LIN {X 0,Y 439.168,Z 450.878,A -85,B 0,C 180,E1 8974.952,E2 8974.952} C_VEL
LIN {X 0,Y 436.814,Z 482.203,A -85,B 0,C 180,E1 8977.325,E2 8977.325} C_VEL
LIN {X 0,Y 434.28,Z 509.002,A -85,B 0,C 180,E1 8980.252,E2 8980.252} C_VEL
LIN {X 0,Y 432.212,Z 531.481,A -85,B 0,C 180,E1 8983.726,E2 8983.726} C_VEL
LIN {X 0,Y 430.436,Z 549.772,A -85,B 0,C 180,E1 8987.816,E2 8987.816} C_VEL
LIN {X 0,Y 429.457,Z 561.558,A -85,B 0,C 180,E1 8991.893,E2 8991.893} C_VEL
LIN {X 0,Y 429.016,Z 568.11,A -85,B 0,C 180,E1 8995.952,E2 8995.952} C_VEL
LIN {X 0,Y 428.83,Z 569.954,A -85,B 0,C 180,E1 8999.999,E2 8999.999} C_VEL
LIN {X 0,Y 428.895,Z 567.151,A -85,B 0,C 180,E1 9004.047,E2 9004.047} C_VEL
LIN {X 0,Y 429.303,Z 559.683,A -85,B 0,C 180,E1 9008.108,E2 9008.108} C_VEL
LIN {X 0,Y 430.114,Z 546.87,A -85,B 0,C 180,E1 9012.191,E2 9012.191} C_VEL
LIN {X 0,Y 431.64,Z 528.884,A -85,B 0,C 180,E1 9016.056,E2 9016.056} C_VEL
LIN {X 0,Y 433.718,Z 505.045,A -85,B 0,C 180,E1 9019.654,E2 9019.654} C_VEL
LIN {X 0,Y 436.275,Z 476.793,A -85,B 0,C 180,E1 9022.668,E2 9022.668} C_VEL
LIN {X 0,Y 438.615,Z 445.158,A -85,B 0,C 180,E1 9025.011,E2 9025.011} C_VEL
LIN {X 0,Y 440.099,Z 410.701,A -85,B 0,C 180,E1 9026.662,E2 9026.662} C_VEL
LIN {X 0,Y 428.142,Z 373.68,A -85,B 0,C 180,E1 9028.308,E2 9028.308} C_VEL
LIN {X 0,Y 427.299,Z 370.16,A -85,B 0,C 180,E1 9028.573,E2 9028.573} C_VEL
LIN {X 0,Y 427.042,Z 370.16,A -85,B 0,C 180,E1 9035.38,E2 9035.38} C_VEL
LIN {X 0,Y 427.064,Z 370.16,A -85,B 0,C 180,E1 9041.893,E2 9041.893} C_VEL
LIN {X 0,Y 427.056,Z 370.16,A -85,B 0,C 180,E1 9048.11,E2 9048.11} C_VEL
LIN {X 0,Y 426.985,Z 370.16,A -85,B 0,C 180,E1 9054.633,E2 9054.633} C_VEL
LIN {X 0,Y 427.166,Z 370.16,A -85,B 0,C 180,E1 9058.611,E2 9058.611} C_VEL
LIN {X 0,Y 444.228,Z 410.083,A -85,B 0,C 180,E1 9061.091,E2 9061.091} C_VEL
LIN {X 0,Y 447.361,Z 421.516,A -85,B 0,C 180,E1 9061.828,E2 9061.828} C_VEL
LIN {X 0,Y 444.469,Z 453.207,A -85,B 0,C 180,E1 9063.532,E2 9063.532} C_VEL
LIN {X 0,Y 440.679,Z 483.869,A -85,B 0,C 180,E1 9066.061,E2 9066.061} C_VEL
LIN {X 0,Y 436.811,Z 510.171,A -85,B 0,C 180,E1 9069.195,E2 9069.195} C_VEL
LIN {X 0,Y 433.382,Z 532.504,A -85,B 0,C 180,E1 9072.992,E2 9072.992} C_VEL
LIN {X 0,Y 430.872,Z 550.061,A -85,B 0,C 180,E1 9077.317,E2 9077.317} C_VEL
LIN {X 0,Y 429.533,Z 561.98,A -85,B 0,C 180,E1 9081.898,E2 9081.898} C_VEL
LIN {X 0,Y 428.963,Z 567.836,A -85,B 0,C 180,E1 9085.955,E2 9085.955} C_VEL
LIN {X 0,Y 428.789,Z 569.7,A -85,B 0,C 180,E1 9090.003,E2 9090.003} C_VEL
LIN {X 0,Y 429.089,Z 566.614,A -85,B 0,C 180,E1 9095.063,E2 9095.063} C_VEL
LIN {X 0,Y 429.816,Z 558.672,A -85,B 0,C 180,E1 9099.531,E2 9099.531} C_VEL
LIN {X 0,Y 431.378,Z 546.18,A -85,B 0,C 180,E1 9103.706,E2 9103.706} C_VEL
LIN {X 0,Y 434.068,Z 528.128,A -85,B 0,C 180,E1 9107.772,E2 9107.772} C_VEL
LIN {X 0,Y 437.501,Z 505.694,A -85,B 0,C 180,E1 9111.319,E2 9111.319} C_VEL
LIN {X 0,Y 441.453,Z 478.009,A -85,B 0,C 180,E1 9114.407,E2 9114.407} C_VEL
LIN {X 0,Y 445.107,Z 446.96,A -85,B 0,C 180,E1 9116.78,E2 9116.78} C_VEL
LIN {X 0,Y 446.908,Z 418.005,A -85,B 0,C 180,E1 9118.269,E2 9118.269} C_VEL
LIN {X 0,Y 433.875,Z 385.514,A -85,B 0,C 180,E1 9120.385,E2 9120.385} C_VEL
LIN {X 0,Y 427.131,Z 370.16,A -85,B 0,C 180,E1 9121.318,E2 9121.318} C_VEL
LIN {X 0,Y 426.919,Z 370.16,A -85,B 0,C 180,E1 9127.078,E2 9127.078} C_VEL
LIN {X 0,Y 426.938,Z 370.16,A -85,B 0,C 180,E1 9132.361,E2 9132.361} C_VEL
LIN {X 0,Y 427.031,Z 370.16,A -85,B 0,C 180,E1 9138.121,E2 9138.121} C_VEL
LIN {X 0,Y 426.934,Z 370.16,A -85,B 0,C 180,E1 9144.651,E2 9144.651} C_VEL
LIN {X 0,Y 427.115,Z 370.16,A -85,B 0,C 180,E1 9150.251,E2 9150.251} C_VEL
LIN {X 0,Y 427.383,Z 370.16,A -85,B 0,C 180,E1 9157.081,E2 9157.081} C_VEL
LIN {X 0,Y 427.621,Z 370.16,A -85,B 0,C 180,E1 9163.549,E2 9163.549} C_VEL
LIN {X 0,Y 427.815,Z 370.16,A -85,B 0,C 180,E1 9169.81,E2 9169.81} C_VEL
LIN {X 0,Y 428.109,Z 370.16,A -85,B 0,C 180,E1 9175.946,E2 9175.946} C_VEL
LIN {X 0,Y 428.238,Z 370.16,A -85,B 0,C 180,E1 9182.027,E2 9182.027} C_VEL
LIN {X 0,Y 427.886,Z 370.16,A -85,B 0,C 180,E1 9188.137,E2 9188.137} C_VEL
LIN {X 0,Y 427.598,Z 370.16,A -85,B 0,C 180,E1 9194.351,E2 9194.351} C_VEL
LIN {X 0,Y 427.412,Z 370.16,A -85,B 0,C 180,E1 9200.746,E2 9200.746} C_VEL
LIN {X 0,Y 427.193,Z 370.16,A -85,B 0,C 180,E1 9207.622,E2 9207.622} C_VEL
LIN {X 0,Y 427.043,Z 370.16,A -85,B 0,C 180,E1 9214.558,E2 9214.558} C_VEL
LIN {X 0,Y 427.042,Z 370.16,A -85,B 0,C 180,E1 9219.653,E2 9219.653} C_VEL
LIN {X 0,Y 427.044,Z 370.16,A -85,B 0,C 180,E1 9225.157,E2 9225.157} C_VEL
LIN {X 0,Y 427.026,Z 370.16,A -85,B 0,C 180,E1 9231.258,E2 9231.258} C_VEL
LIN {X 0,Y 427.065,Z 370.71,A -85,B 0,C 180,E1 9233.504,E2 9233.504} C_VEL
LIN {X 0,Y 445.595,Z 414.881,A -85,B 0,C 180,E1 9235.972,E2 9235.972} C_VEL
LIN {X 0,Y 448.263,Z 424.22,A -85,B 0,C 180,E1 9236.409,E2 9236.409} C_VEL
LIN {X 0,Y 445.751,Z 460.729,A -85,B 0,C 180,E1 9237.649,E2 9237.649} C_VEL
LIN {X 0,Y 442.346,Z 497.11,A -85,B 0,C 180,E1 9239.677,E2 9239.677} C_VEL
LIN {X 0,Y 438.45,Z 531.769,A -85,B 0,C 180,E1 9242.523,E2 9242.523} C_VEL
LIN {X 0,Y 435.416,Z 557.233,A -85,B 0,C 180,E1 9245.338,E2 9245.338} C_VEL
LIN {X 0,Y 430.206,Z 569.543,A -85,B 0,C 180,E1 9246.847,E2 9246.847} C_VEL
LIN {X 0,Y 425.037,Z 580.954,A -85,B 0,C 180,E1 9248.491,E2 9248.491} C_VEL
LIN {X 0,Y 422.611,Z 603.04,A -85,B 0,C 180,E1 9252.815,E2 9252.815} C_VEL
LIN {X 0,Y 421.281,Z 620.303,A -85,B 0,C 180,E1 9257.545,E2 9257.545} C_VEL
LIN {X 0,Y 420.847,Z 630.496,A -85,B 0,C 180,E1 9261.724,E2 9261.724} C_VEL
LIN {X 0,Y 420.642,Z 636.421,A -85,B 0,C 180,E1 9265.869,E2 9265.869} C_VEL
LIN {X 0,Y 420.644,Z 638.428,A -85,B 0,C 180,E1 9269.997,E2 9269.997} C_VEL
LIN {X 0,Y 420.633,Z 636.423,A -85,B 0,C 180,E1 9274.125,E2 9274.125} C_VEL
LIN {X 0,Y 420.896,Z 629.4,A -85,B 0,C 180,E1 9278.824,E2 9278.824} C_VEL
LIN {X 0,Y 421.612,Z 616.155,A -85,B 0,C 180,E1 9283.774,E2 9283.774} C_VEL
LIN {X 0,Y 423.23,Z 597.024,A -85,B 0,C 180,E1 9288.502,E2 9288.502} C_VEL
LIN {X 0,Y 425.888,Z 572.969,A -85,B 0,C 180,E1 9292.795,E2 9292.795} C_VEL
LIN {X 0,Y 429.597,Z 543.692,A -85,B 0,C 180,E1 9296.624,E2 9296.624} C_VEL
LIN {X 0,Y 433.587,Z 511.563,A -85,B 0,C 180,E1 9299.691,E2 9299.691} C_VEL
LIN {X 0,Y 437.479,Z 476.127,A -85,B 0,C 180,E1 9302.084,E2 9302.084} C_VEL
LIN {X 0,Y 440.522,Z 439.527,A -85,B 0,C 180,E1 9303.673,E2 9303.673} C_VEL
LIN {X 0,Y 440.953,Z 423.155,A -85,B 0,C 180,E1 9304.186,E2 9304.186} C_VEL
LIN {X 0,Y 426.757,Z 387.404,A -85,B 0,C 180,E1 9306.172,E2 9306.172} C_VEL
LIN {X 0,Y 419.113,Z 370.16,A -85,B 0,C 180,E1 9307.373,E2 9307.373} C_VEL
LIN {X 0,Y 418.883,Z 370.16,A -85,B 0,C 180,E1 9313.709,E2 9313.709} C_VEL
LIN {X 0,Y 418.918,Z 370.16,A -85,B 0,C 180,E1 9319.419,E2 9319.419} C_VEL
LIN {X 0,Y 419.043,Z 370.16,A -85,B 0,C 180,E1 9326.191,E2 9326.191} C_VEL
LIN {X 0,Y 419.24,Z 370.16,A -85,B 0,C 180,E1 9330.068,E2 9330.068} C_VEL
LIN {X 0,Y 431.504,Z 401.917,A -85,B 0,C 180,E1 9332.061,E2 9332.061} C_VEL
LIN {X 0,Y 434.096,Z 415.976,A -85,B 0,C 180,E1 9332.758,E2 9332.758} C_VEL
LIN {X 0,Y 432.14,Z 450.362,A -85,B 0,C 180,E1 9334.422,E2 9334.422} C_VEL
LIN {X 0,Y 429.68,Z 481.926,A -85,B 0,C 180,E1 9336.818,E2 9336.818} C_VEL
LIN {X 0,Y 426.891,Z 509.818,A -85,B 0,C 180,E1 9339.895,E2 9339.895} C_VEL
LIN {X 0,Y 424.648,Z 532.264,A -85,B 0,C 180,E1 9343.427,E2 9343.427} C_VEL
LIN {X 0,Y 422.86,Z 548.653,A -85,B 0,C 180,E1 9347.069,E2 9347.069} C_VEL
LIN {X 0,Y 421.801,Z 560.776,A -85,B 0,C 180,E1 9351.052,E2 9351.052} C_VEL
LIN {X 0,Y 421.254,Z 567.704,A -85,B 0,C 180,E1 9354.844,E2 9354.844} C_VEL
LIN {X 0,Y 421.103,Z 570.276,A -85,B 0,C 180,E1 9357.938,E2 9357.938} C_VEL
LIN {X 0,Y 420.875,Z 569.759,A -85,B 0,C 180,E1 9362.06,E2 9362.06} C_VEL
LIN {X 0,Y 421.239,Z 563.556,A -85,B 0,C 180,E1 9366.706,E2 9366.706} C_VEL
LIN {X 0,Y 421.863,Z 552.754,A -85,B 0,C 180,E1 9370.858,E2 9370.858} C_VEL
LIN {X 0,Y 423.299,Z 535.645,A -85,B 0,C 180,E1 9375.072,E2 9375.072} C_VEL
LIN {X 0,Y 425.417,Z 512.927,A -85,B 0,C 180,E1 9378.922,E2 9378.922} C_VEL
LIN {X 0,Y 427.842,Z 486.703,A -85,B 0,C 180,E1 9382.082,E2 9382.082} C_VEL
LIN {X 0,Y 430.546,Z 455.568,A -85,B 0,C 180,E1 9384.714,E2 9384.714} C_VEL
LIN {X 0,Y 432.733,Z 422.031,A -85,B 0,C 180,E1 9386.586,E2 9386.586} C_VEL
LIN {X 0,Y 432.099,Z 410.056,A -85,B 0,C 180,E1 9387.118,E2 9387.118} C_VEL
LIN {X 0,Y 419.359,Z 370.16,A -85,B 0,C 180,E1 9388.913,E2 9388.913} C_VEL
LIN {X 0,Y 419.152,Z 370.16,A -85,B 0,C 180,E1 9395.301,E2 9395.301} C_VEL
LIN {X 0,Y 419.087,Z 370.16,A -85,B 0,C 180,E1 9400.663,E2 9400.663} C_VEL
LIN {X 0,Y 419.058,Z 370.16,A -85,B 0,C 180,E1 9406.657,E2 9406.657} C_VEL
LIN {X 0,Y 419.088,Z 370.16,A -85,B 0,C 180,E1 9412.627,E2 9412.627} C_VEL
LIN {X 0,Y 419.241,Z 370.651,A -85,B 0,C 180,E1 9417.915,E2 9417.915} C_VEL
LIN {X 0,Y 435.983,Z 408.61,A -85,B 0,C 180,E1 9420.361,E2 9420.361} C_VEL
LIN {X 0,Y 440.461,Z 423.194,A -85,B 0,C 180,E1 9421.364,E2 9421.364} C_VEL
LIN {X 0,Y 437.323,Z 455.539,A -85,B 0,C 180,E1 9423.161,E2 9423.161} C_VEL
LIN {X 0,Y 433.514,Z 484.713,A -85,B 0,C 180,E1 9425.64,E2 9425.64} C_VEL
LIN {X 0,Y 429.389,Z 511.291,A -85,B 0,C 180,E1 9428.871,E2 9428.871} C_VEL
LIN {X 0,Y 425.827,Z 533.214,A -85,B 0,C 180,E1 9432.68,E2 9432.68} C_VEL
LIN {X 0,Y 423.148,Z 550.734,A -85,B 0,C 180,E1 9437.082,E2 9437.082} C_VEL
LIN {X 0,Y 421.712,Z 562.634,A -85,B 0,C 180,E1 9441.747,E2 9441.747} C_VEL
LIN {X 0,Y 421.099,Z 568.476,A -85,B 0,C 180,E1 9445.88,E2 9445.88} C_VEL
LIN {X 0,Y 420.93,Z 570.336,A -85,B 0,C 180,E1 9450.003,E2 9450.003} C_VEL
LIN {X 0,Y 421.229,Z 567.258,A -85,B 0,C 180,E1 9455.158,E2 9455.158} C_VEL
LIN {X 0,Y 422.022,Z 559.446,A -85,B 0,C 180,E1 9459.661,E2 9459.661} C_VEL
LIN {X 0,Y 423.69,Z 546.865,A -85,B 0,C 180,E1 9463.96,E2 9463.96} C_VEL
LIN {X 0,Y 426.55,Z 528.856,A -85,B 0,C 180,E1 9468.096,E2 9468.096} C_VEL
LIN {X 0,Y 430.179,Z 506.541,A -85,B 0,C 180,E1 9471.69,E2 9471.69} C_VEL
LIN {X 0,Y 434.313,Z 478.921,A -85,B 0,C 180,E1 9474.833,E2 9474.833} C_VEL
LIN {X 0,Y 438.149,Z 448.064,A -85,B 0,C 180,E1 9477.24,E2 9477.24} C_VEL
LIN {X 0,Y 439.911,Z 420.118,A -85,B 0,C 180,E1 9478.737,E2 9478.737} C_VEL
LIN {X 0,Y 427.218,Z 387.979,A -85,B 0,C 180,E1 9480.916,E2 9480.916} C_VEL
LIN {X 0,Y 419.198,Z 370.16,A -85,B 0,C 180,E1 9482.049,E2 9482.049} C_VEL
LIN {X 0,Y 419.008,Z 370.16,A -85,B 0,C 180,E1 9487.9,E2 9487.9} C_VEL
LIN {X 0,Y 418.98,Z 370.16,A -85,B 0,C 180,E1 9493.727,E2 9493.727} C_VEL
LIN {X 0,Y 419.04,Z 370.16,A -85,B 0,C 180,E1 9499.437,E2 9499.437} C_VEL
LIN {X 0,Y 419.027,Z 370.16,A -85,B 0,C 180,E1 9506.205,E2 9506.205} C_VEL
LIN {X 0,Y 419.239,Z 370.16,A -85,B 0,C 180,E1 9512.004,E2 9512.004} C_VEL
LIN {X 0,Y 419.51,Z 370.16,A -85,B 0,C 180,E1 9518.848,E2 9518.848} C_VEL
LIN {X 0,Y 419.768,Z 370.16,A -85,B 0,C 180,E1 9525.378,E2 9525.378} C_VEL
LIN {X 0,Y 419.955,Z 370.16,A -85,B 0,C 180,E1 9531.711,E2 9531.711} C_VEL
LIN {X 0,Y 420.185,Z 370.16,A -85,B 0,C 180,E1 9537.937,E2 9537.937} C_VEL
LIN {X 0,Y 420.066,Z 370.16,A -85,B 0,C 180,E1 9544.135,E2 9544.135} C_VEL
LIN {X 0,Y 419.817,Z 370.16,A -85,B 0,C 180,E1 9550.389,E2 9550.389} C_VEL
LIN {X 0,Y 419.642,Z 370.16,A -85,B 0,C 180,E1 9556.776,E2 9556.776} C_VEL
LIN {X 0,Y 419.398,Z 370.16,A -85,B 0,C 180,E1 9563.396,E2 9563.396} C_VEL
LIN {X 0,Y 419.188,Z 370.16,A -85,B 0,C 180,E1 9570.374,E2 9570.374} C_VEL
LIN {X 0,Y 419.117,Z 370.16,A -85,B 0,C 180,E1 9577.37,E2 9577.37} C_VEL
LIN {X 0,Y 419.041,Z 370.16,A -85,B 0,C 180,E1 9583.729,E2 9583.729} C_VEL
LIN {X 0,Y 419.061,Z 370.16,A -85,B 0,C 180,E1 9589.433,E2 9589.433} C_VEL
LIN {X 0,Y 419.107,Z 370.799,A -85,B 0,C 180,E1 9592.779,E2 9592.779} C_VEL
LIN {X 0,Y 437.415,Z 413.266,A -85,B 0,C 180,E1 9595.287,E2 9595.287} C_VEL
LIN {X 0,Y 441.354,Z 426.137,A -85,B 0,C 180,E1 9595.939,E2 9595.939} C_VEL
LIN {X 0,Y 438.727,Z 462.019,A -85,B 0,C 180,E1 9597.211,E2 9597.211} C_VEL
LIN {X 0,Y 435.147,Z 497.819,A -85,B 0,C 180,E1 9599.266,E2 9599.266} C_VEL
LIN {X 0,Y 431.048,Z 531.883,A -85,B 0,C 180,E1 9602.133,E2 9602.133} C_VEL
LIN {X 0,Y 427.258,Z 562.326,A -85,B 0,C 180,E1 9605.671,E2 9605.671} C_VEL
LIN {X 0,Y 425.037,Z 580.954,A -85,B 0,C 180,E1 9608.491,E2 9608.491} C_VEL
LIN {X 0,Y 419.96,Z 591.453,A -85,B 0,C 180,E1 9610.27,E2 9610.27} C_VEL
LIN {X 0,Y 415.012,Z 600.931,A -85,B 0,C 180,E1 9612.178,E2 9612.178} C_VEL
LIN {X 0,Y 413.544,Z 618.3,A -85,B 0,C 180,E1 9616.898,E2 9616.898} C_VEL
LIN {X 0,Y 412.968,Z 630.279,A -85,B 0,C 180,E1 9621.818,E2 9621.818} C_VEL
LIN {X 0,Y 412.764,Z 635.764,A -85,B 0,C 180,E1 9625.79,E2 9625.79} C_VEL
LIN {X 0,Y 412.769,Z 637.791,A -85,B 0,C 180,E1 9629.997,E2 9629.997} C_VEL
LIN {X 0,Y 412.753,Z 635.77,A -85,B 0,C 180,E1 9634.204,E2 9634.204} C_VEL
LIN {X 0,Y 413.006,Z 628.758,A -85,B 0,C 180,E1 9638.959,E2 9638.959} C_VEL
LIN {X 0,Y 413.751,Z 615.794,A -85,B 0,C 180,E1 9643.917,E2 9643.917} C_VEL
LIN {X 0,Y 415.385,Z 597.315,A -85,B 0,C 180,E1 9648.628,E2 9648.628} C_VEL
LIN {X 0,Y 418.192,Z 573.458,A -85,B 0,C 180,E1 9653.015,E2 9653.015} C_VEL
LIN {X 0,Y 422.173,Z 543.785,A -85,B 0,C 180,E1 9657.006,E2 9657.006} C_VEL
LIN {X 0,Y 426.35,Z 512.102,A -85,B 0,C 180,E1 9660.1,E2 9660.1} C_VEL
LIN {X 0,Y 430.36,Z 477.549,A -85,B 0,C 180,E1 9662.502,E2 9662.502} C_VEL
LIN {X 0,Y 433.615,Z 440.992,A -85,B 0,C 180,E1 9664.155,E2 9664.155} C_VEL
LIN {X 0,Y 434.123,Z 425.328,A -85,B 0,C 180,E1 9664.664,E2 9664.664} C_VEL
LIN {X 0,Y 420.847,Z 391.503,A -85,B 0,C 180,E1 9666.614,E2 9666.614} C_VEL
LIN {X 0,Y 411.148,Z 370.16,A -85,B 0,C 180,E1 9668.109,E2 9668.109} C_VEL
LIN {X 0,Y 410.912,Z 370.16,A -85,B 0,C 180,E1 9675.57,E2 9675.57} C_VEL
LIN {X 0,Y 410.97,Z 370.16,A -85,B 0,C 180,E1 9681.225,E2 9681.225} C_VEL
LIN {X 0,Y 411.155,Z 370.16,A -85,B 0,C 180,E1 9687.869,E2 9687.869} C_VEL
LIN {X 0,Y 411.244,Z 370.363,A -85,B 0,C 180,E1 9689.219,E2 9689.219} C_VEL
LIN {X 0,Y 423.804,Z 400.867,A -85,B 0,C 180,E1 9691.385,E2 9691.385} C_VEL
LIN {X 0,Y 427.245,Z 417.052,A -85,B 0,C 180,E1 9692.258,E2 9692.258} C_VEL
LIN {X 0,Y 425.085,Z 451.803,A -85,B 0,C 180,E1 9693.99,E2 9693.99} C_VEL
LIN {X 0,Y 422.486,Z 482.835,A -85,B 0,C 180,E1 9696.399,E2 9696.399} C_VEL
LIN {X 0,Y 419.645,Z 509.505,A -85,B 0,C 180,E1 9699.364,E2 9699.364} C_VEL
LIN {X 0,Y 417.231,Z 531.696,A -85,B 0,C 180,E1 9702.852,E2 9702.852} C_VEL
LIN {X 0,Y 415.179,Z 549.482,A -85,B 0,C 180,E1 9706.825,E2 9706.825} C_VEL
LIN {X 0,Y 414.023,Z 561.46,A -85,B 0,C 180,E1 9710.835,E2 9710.835} C_VEL
LIN {X 0,Y 413.414,Z 568.464,A -85,B 0,C 180,E1 9714.746,E2 9714.746} C_VEL
LIN {X 0,Y 413.253,Z 570.988,A -85,B 0,C 180,E1 9717.899,E2 9717.899} C_VEL
LIN {X 0,Y 413.002,Z 570.394,A -85,B 0,C 180,E1 9722.099,E2 9722.099} C_VEL
LIN {X 0,Y 413.381,Z 564.063,A -85,B 0,C 180,E1 9726.834,E2 9726.834} C_VEL
LIN {X 0,Y 414.072,Z 553.085,A -85,B 0,C 180,E1 9731.065,E2 9731.065} C_VEL
LIN {X 0,Y 415.601,Z 535.785,A -85,B 0,C 180,E1 9735.358,E2 9735.358} C_VEL
LIN {X 0,Y 417.81,Z 512.827,A -85,B 0,C 180,E1 9739.271,E2 9739.271} C_VEL
LIN {X 0,Y 420.411,Z 486.124,A -85,B 0,C 180,E1 9742.494,E2 9742.494} C_VEL
LIN {X 0,Y 423.186,Z 455.014,A -85,B 0,C 180,E1 9745.124,E2 9745.124} C_VEL
LIN {X 0,Y 425.374,Z 421.762,A -85,B 0,C 180,E1 9746.988,E2 9746.988} C_VEL
LIN {X 0,Y 424.711,Z 411.849,A -85,B 0,C 180,E1 9747.448,E2 9747.448} C_VEL
LIN {X 0,Y 411.414,Z 370.16,A -85,B 0,C 180,E1 9749.377,E2 9749.377} C_VEL
LIN {X 0,Y 411.2,Z 370.16,A -85,B 0,C 180,E1 9756.089,E2 9756.089} C_VEL
LIN {X 0,Y 411.095,Z 370.16,A -85,B 0,C 180,E1 9762.568,E2 9762.568} C_VEL
LIN {X 0,Y 411.079,Z 370.16,A -85,B 0,C 180,E1 9768.482,E2 9768.482} C_VEL
LIN {X 0,Y 411.14,Z 370.16,A -85,B 0,C 180,E1 9774.102,E2 9774.102} C_VEL
LIN {X 0,Y 411.206,Z 370.16,A -85,B 0,C 180,E1 9777.119,E2 9777.119} C_VEL
LIN {X 0,Y 419.182,Z 387.551,A -85,B 0,C 180,E1 9778.238,E2 9778.238} C_VEL
LIN {X 0,Y 432.089,Z 419.327,A -85,B 0,C 180,E1 9780.483,E2 9780.483} C_VEL
LIN {X 0,Y 433.443,Z 426.992,A -85,B 0,C 180,E1 9780.982,E2 9780.982} C_VEL
LIN {X 0,Y 429.994,Z 459.468,A -85,B 0,C 180,E1 9782.906,E2 9782.906} C_VEL
LIN {X 0,Y 425.816,Z 489.229,A -85,B 0,C 180,E1 9785.59,E2 9785.59} C_VEL
LIN {X 0,Y 421.51,Z 515.071,A -85,B 0,C 180,E1 9788.954,E2 9788.954} C_VEL
LIN {X 0,Y 417.89,Z 536.392,A -85,B 0,C 180,E1 9792.885,E2 9792.885} C_VEL
LIN {X 0,Y 415.207,Z 553.032,A -85,B 0,C 180,E1 9797.366,E2 9797.366} C_VEL
LIN {X 0,Y 413.907,Z 563.286,A -85,B 0,C 180,E1 9801.59,E2 9801.59} C_VEL
LIN {X 0,Y 413.257,Z 569.115,A -85,B 0,C 180,E1 9805.801,E2 9805.801} C_VEL
LIN {X 0,Y 413.056,Z 570.973,A -85,B 0,C 180,E1 9810.003,E2 9810.003} C_VEL
LIN {X 0,Y 413.393,Z 567.899,A -85,B 0,C 180,E1 9815.256,E2 9815.256} C_VEL
LIN {X 0,Y 414.199,Z 560.429,A -85,B 0,C 180,E1 9819.708,E2 9819.708} C_VEL
LIN {X 0,Y 416.007,Z 547.547,A -85,B 0,C 180,E1 9824.223,E2 9824.223} C_VEL
LIN {X 0,Y 419.041,Z 529.58,A -85,B 0,C 180,E1 9828.432,E2 9828.432} C_VEL
LIN {X 0,Y 422.868,Z 507.311,A -85,B 0,C 180,E1 9832.084,E2 9832.084} C_VEL
LIN {X 0,Y 427.203,Z 479.741,A -85,B 0,C 180,E1 9835.282,E2 9835.282} C_VEL
LIN {X 0,Y 431.171,Z 449.496,A -85,B 0,C 180,E1 9837.689,E2 9837.689} C_VEL
LIN {X 0,Y 433.265,Z 423.226,A -85,B 0,C 180,E1 9839.13,E2 9839.13} C_VEL
LIN {X 0,Y 420.863,Z 391.278,A -85,B 0,C 180,E1 9841.421,E2 9841.421} C_VEL
LIN {X 0,Y 411.17,Z 370.16,A -85,B 0,C 180,E1 9842.883,E2 9842.883} C_VEL
LIN {X 0,Y 410.992,Z 370.16,A -85,B 0,C 180,E1 9849.329,E2 9849.329} C_VEL
LIN {X 0,Y 411.051,Z 370.16,A -85,B 0,C 180,E1 9855.593,E2 9855.593} C_VEL
LIN {X 0,Y 411.046,Z 370.16,A -85,B 0,C 180,E1 9861.237,E2 9861.237} C_VEL
LIN {X 0,Y 411.126,Z 370.16,A -85,B 0,C 180,E1 9867.888,E2 9867.888} C_VEL
LIN {X 0,Y 411.354,Z 370.16,A -85,B 0,C 180,E1 9873.793,E2 9873.793} C_VEL
LIN {X 0,Y 411.651,Z 370.16,A -85,B 0,C 180,E1 9880.673,E2 9880.673} C_VEL
LIN {X 0,Y 411.904,Z 370.16,A -85,B 0,C 180,E1 9887.262,E2 9887.262} C_VEL
LIN {X 0,Y 412.089,Z 370.16,A -85,B 0,C 180,E1 9893.674,E2 9893.674} C_VEL
LIN {X 0,Y 412.422,Z 370.16,A -85,B 0,C 180,E1 9900.001,E2 9900.001} C_VEL
LIN {X 0,Y 412.057,Z 370.16,A -85,B 0,C 180,E1 9907.227,E2 9907.227} C_VEL
LIN {X 0,Y 411.826,Z 370.16,A -85,B 0,C 180,E1 9912.744,E2 9912.744} C_VEL
LIN {X 0,Y 411.623,Z 370.16,A -85,B 0,C 180,E1 9919.332,E2 9919.332} C_VEL
LIN {X 0,Y 411.359,Z 370.16,A -85,B 0,C 180,E1 9926.209,E2 9926.209} C_VEL
LIN {X 0,Y 411.197,Z 370.16,A -85,B 0,C 180,E1 9933.524,E2 9933.524} C_VEL
LIN {X 0,Y 411.089,Z 370.16,A -85,B 0,C 180,E1 9939.337,E2 9939.337} C_VEL
LIN {X 0,Y 411.085,Z 370.16,A -85,B 0,C 180,E1 9945.591,E2 9945.591} C_VEL
LIN {X 0,Y 411.206,Z 370.844,A -85,B 0,C 180,E1 9952.023,E2 9952.023} C_VEL
LIN {X 0,Y 430.74,Z 415.558,A -85,B 0,C 180,E1 9954.792,E2 9954.792} C_VEL
LIN {X 0,Y 434.427,Z 429.233,A -85,B 0,C 180,E1 9955.486,E2 9955.486} C_VEL
LIN {X 0,Y 431.365,Z 467.198,A -85,B 0,C 180,E1 9956.948,E2 9956.948} C_VEL
LIN {X 0,Y 427.553,Z 501.976,A -85,B 0,C 180,E1 9959.104,E2 9959.104} C_VEL
LIN {X 0,Y 423.301,Z 535.443,A -85,B 0,C 180,E1 9962.079,E2 9962.079} C_VEL
LIN {X 0,Y 419.27,Z 565.21,A -85,B 0,C 180,E1 9965.746,E2 9965.746} C_VEL
LIN {X 0,Y 416.082,Z 590.906,A -85,B 0,C 180,E1 9970.052,E2 9970.052} C_VEL
LIN {X 0,Y 415.012,Z 600.931,A -85,B 0,C 180,E1 9972.178,E2 9972.178} C_VEL
LIN {X 0,Y 413.333,Z 605.378,A -85,B 0,C 180,E1 9973.203,E2 9973.203} C_VEL
LIN {X 0,Y 405.931,Z 615.887,A -85,B 0,C 180,E1 9976.077,E2 9976.077} C_VEL
LIN {X 0,Y 405.797,Z 616.736,A -85,B 0,C 180,E1 9976.362,E2 9976.362} C_VEL
LIN {X 0,Y 405.089,Z 629.102,A -85,B 0,C 180,E1 9981.399,E2 9981.399} C_VEL
LIN {X 0,Y 404.909,Z 635.116,A -85,B 0,C 180,E1 9985.708,E2 9985.708} C_VEL
LIN {X 0,Y 404.893,Z 637.154,A -85,B 0,C 180,E1 9989.997,E2 9989.997} C_VEL
LIN {X 0,Y 404.898,Z 635.122,A -85,B 0,C 180,E1 9994.285,E2 9994.285} C_VEL
LIN {X 0,Y 405.113,Z 628.072,A -85,B 0,C 180,E1 9999.135,E2 9999.135} C_VEL
LIN {X 0,Y 405.876,Z 615.307,A -85,B 0,C 180,E1 10004.113,E2 10004.113} C_VEL
LIN {X 0,Y 407.587,Z 597.238,A -85,B 0,C 180,E1 10008.843,E2 10008.843} C_VEL
LIN {X 0,Y 410.576,Z 573.342,A -85,B 0,C 180,E1 10013.346,E2 10013.346} C_VEL
LIN {X 0,Y 414.648,Z 544.81,A -85,B 0,C 180,E1 10017.298,E2 10017.298} C_VEL
LIN {X 0,Y 419.122,Z 512.664,A -85,B 0,C 180,E1 10020.524,E2 10020.524} C_VEL
LIN {X 0,Y 423.188,Z 479.368,A -85,B 0,C 180,E1 10022.91,E2 10022.91} C_VEL
LIN {X 0,Y 426.737,Z 442.585,A -85,B 0,C 180,E1 10024.649,E2 10024.649} C_VEL
LIN {X 0,Y 427.113,Z 426.736,A -85,B 0,C 180,E1 10025.2,E2 10025.2} C_VEL
LIN {X 0,Y 414.349,Z 394.294,A -85,B 0,C 180,E1 10027.157,E2 10027.157} C_VEL
LIN {X 0,Y 403.169,Z 370.16,A -85,B 0,C 180,E1 10028.865,E2 10028.865} C_VEL
LIN {X 0,Y 403.011,Z 370.16,A -85,B 0,C 180,E1 10035.536,E2 10035.536} C_VEL
LIN {X 0,Y 403.015,Z 370.16,A -85,B 0,C 180,E1 10042.075,E2 10042.075} C_VEL
LIN {X 0,Y 403.277,Z 370.693,A -85,B 0,C 180,E1 10048.257,E2 10048.257} C_VEL
LIN {X 0,Y 415.423,Z 397.776,A -85,B 0,C 180,E1 10050.512,E2 10050.512} C_VEL
LIN {X 0,Y 420.475,Z 418.065,A -85,B 0,C 180,E1 10051.725,E2 10051.725} C_VEL
LIN {X 0,Y 418.119,Z 453.08,A -85,B 0,C 180,E1 10053.516,E2 10053.516} C_VEL
LIN {X 0,Y 415.166,Z 485.313,A -85,B 0,C 180,E1 10056.099,E2 10056.099} C_VEL
LIN {X 0,Y 412.063,Z 512.481,A -85,B 0,C 180,E1 10059.259,E2 10059.259} C_VEL
LIN {X 0,Y 409.547,Z 534.033,A -85,B 0,C 180,E1 10062.798,E2 10062.798} C_VEL
LIN {X 0,Y 407.492,Z 550.363,A -85,B 0,C 180,E1 10066.572,E2 10066.572} C_VEL
LIN {X 0,Y 406.234,Z 562.298,A -85,B 0,C 180,E1 10070.658,E2 10070.658} C_VEL
LIN {X 0,Y 405.591,Z 569.237,A -85,B 0,C 180,E1 10074.644,E2 10074.644} C_VEL
LIN {X 0,Y 405.392,Z 571.705,A -85,B 0,C 180,E1 10077.858,E2 10077.858} C_VEL
LIN {X 0,Y 405.13,Z 571.023,A -85,B 0,C 180,E1 10082.14,E2 10082.14} C_VEL
LIN {X 0,Y 405.554,Z 564.535,A -85,B 0,C 180,E1 10086.967,E2 10086.967} C_VEL
LIN {X 0,Y 406.266,Z 553.368,A -85,B 0,C 180,E1 10091.28,E2 10091.28} C_VEL
LIN {X 0,Y 407.893,Z 536.063,A -85,B 0,C 180,E1 10095.608,E2 10095.608} C_VEL
LIN {X 0,Y 410.173,Z 513.054,A -85,B 0,C 180,E1 10099.574,E2 10099.574} C_VEL
LIN {X 0,Y 412.968,Z 485.493,A -85,B 0,C 180,E1 10102.922,E2 10102.922} C_VEL
LIN {X 0,Y 415.846,Z 453.985,A -85,B 0,C 180,E1 10105.584,E2 10105.584} C_VEL
LIN {X 0,Y 418.149,Z 420.154,A -85,B 0,C 180,E1 10107.459,E2 10107.459} C_VEL
LIN {X 0,Y 414.873,Z 404.841,A -85,B 0,C 180,E1 10108.265,E2 10108.265} C_VEL
LIN {X 0,Y 403.48,Z 370.16,A -85,B 0,C 180,E1 10109.921,E2 10109.921} C_VEL
LIN {X 0,Y 403.18,Z 370.16,A -85,B 0,C 180,E1 10116.924,E2 10116.924} C_VEL
LIN {X 0,Y 403.193,Z 370.16,A -85,B 0,C 180,E1 10122.519,E2 10122.519} C_VEL
LIN {X 0,Y 403.155,Z 370.16,A -85,B 0,C 180,E1 10128.677,E2 10128.677} C_VEL
LIN {X 0,Y 403.27,Z 370.16,A -85,B 0,C 180,E1 10136.295,E2 10136.295} C_VEL
LIN {X 0,Y 420.982,Z 409.687,A -85,B 0,C 180,E1 10139.089,E2 10139.089} C_VEL
LIN {X 0,Y 426.621,Z 428.304,A -85,B 0,C 180,E1 10140.473,E2 10140.473} C_VEL
LIN {X 0,Y 423.045,Z 460.42,A -85,B 0,C 180,E1 10142.424,E2 10142.424} C_VEL
LIN {X 0,Y 418.678,Z 490.059,A -85,B 0,C 180,E1 10145.146,E2 10145.146} C_VEL
LIN {X 0,Y 414.141,Z 515.812,A -85,B 0,C 180,E1 10148.561,E2 10148.561} C_VEL
LIN {X 0,Y 410.321,Z 537.084,A -85,B 0,C 180,E1 10152.559,E2 10152.559} C_VEL
LIN {X 0,Y 407.477,Z 553.701,A -85,B 0,C 180,E1 10157.123,E2 10157.123} C_VEL
LIN {X 0,Y 406.076,Z 563.939,A -85,B 0,C 180,E1 10161.427,E2 10161.427} C_VEL
LIN {X 0,Y 405.394,Z 569.755,A -85,B 0,C 180,E1 10165.72,E2 10165.72} C_VEL
LIN {X 0,Y 405.191,Z 571.61,A -85,B 0,C 180,E1 10170.003,E2 10170.003} C_VEL
LIN {X 0,Y 405.533,Z 568.542,A -85,B 0,C 180,E1 10175.358,E2 10175.358} C_VEL
LIN {X 0,Y 406.465,Z 560.699,A -85,B 0,C 180,E1 10180.063,E2 10180.063} C_VEL
LIN {X 0,Y 408.329,Z 548.225,A -85,B 0,C 180,E1 10184.496,E2 10184.496} C_VEL
LIN {X 0,Y 411.547,Z 530.298,A -85,B 0,C 180,E1 10188.78,E2 10188.78} C_VEL
LIN {X 0,Y 415.578,Z 508.075,A -85,B 0,C 180,E1 10192.493,E2 10192.493} C_VEL
LIN {X 0,Y 420.106,Z 480.748,A -85,B 0,C 180,E1 10195.726,E2 10195.726} C_VEL
LIN {X 0,Y 424.262,Z 450.521,A -85,B 0,C 180,E1 10198.18,E2 10198.18} C_VEL
LIN {X 0,Y 426.475,Z 425.738,A -85,B 0,C 180,E1 10199.576,E2 10199.576} C_VEL
LIN {X 0,Y 414.227,Z 393.643,A -85,B 0,C 180,E1 10201.986,E2 10201.986} C_VEL
LIN {X 0,Y 403.241,Z 370.16,A -85,B 0,C 180,E1 10203.704,E2 10203.704} C_VEL
LIN {X 0,Y 403.056,Z 370.16,A -85,B 0,C 180,E1 10211.306,E2 10211.306} C_VEL
LIN {X 0,Y 403.154,Z 370.16,A -85,B 0,C 180,E1 10217.476,E2 10217.476} C_VEL
LIN {X 0,Y 403.081,Z 370.16,A -85,B 0,C 180,E1 10223.065,E2 10223.065} C_VEL
LIN {X 0,Y 403.235,Z 370.16,A -85,B 0,C 180,E1 10229.721,E2 10229.721} C_VEL
LIN {X 0,Y 403.47,Z 370.16,A -85,B 0,C 180,E1 10235.624,E2 10235.624} C_VEL
LIN {X 0,Y 403.805,Z 370.16,A -85,B 0,C 180,E1 10242.548,E2 10242.548} C_VEL
LIN {X 0,Y 404.021,Z 370.16,A -85,B 0,C 180,E1 10249.203,E2 10249.203} C_VEL
LIN {X 0,Y 404.35,Z 370.16,A -85,B 0,C 180,E1 10255.707,E2 10255.707} C_VEL
LIN {X 0,Y 404.515,Z 370.16,A -85,B 0,C 180,E1 10262.146,E2 10262.146} C_VEL
LIN {X 0,Y 404.103,Z 370.16,A -85,B 0,C 180,E1 10268.62,E2 10268.62} C_VEL
LIN {X 0,Y 403.806,Z 370.16,A -85,B 0,C 180,E1 10275.216,E2 10275.216} C_VEL
LIN {X 0,Y 403.584,Z 370.16,A -85,B 0,C 180,E1 10282.033,E2 10282.033} C_VEL
LIN {X 0,Y 403.312,Z 370.16,A -85,B 0,C 180,E1 10289.209,E2 10289.209} C_VEL
LIN {X 0,Y 403.236,Z 370.16,A -85,B 0,C 180,E1 10294.307,E2 10294.307} C_VEL
LIN {X 0,Y 403.15,Z 370.16,A -85,B 0,C 180,E1 10301.314,E2 10301.314} C_VEL
LIN {X 0,Y 403.175,Z 370.16,A -85,B 0,C 180,E1 10307.471,E2 10307.471} C_VEL
LIN {X 0,Y 403.172,Z 370.16,A -85,B 0,C 180,E1 10311.194,E2 10311.194} C_VEL
LIN {X 0,Y 424.127,Z 417.995,A -85,B 0,C 180,E1 10314.287,E2 10314.287} C_VEL
LIN {X 0,Y 427.634,Z 430.383,A -85,B 0,C 180,E1 10314.965,E2 10314.965} C_VEL
LIN {X 0,Y 424.458,Z 467.413,A -85,B 0,C 180,E1 10316.434,E2 10316.434} C_VEL
LIN {X 0,Y 420.385,Z 502.647,A -85,B 0,C 180,E1 10318.668,E2 10318.668} C_VEL
LIN {X 0,Y 415.864,Z 536.357,A -85,B 0,C 180,E1 10321.751,E2 10321.751} C_VEL
LIN {X 0,Y 411.55,Z 566.2,A -85,B 0,C 180,E1 10325.55,E2 10325.55} C_VEL
LIN {X 0,Y 408.26,Z 591.512,A -85,B 0,C 180,E1 10329.936,E2 10329.936} C_VEL
LIN {X 0,Y 406.11,Z 611.897,A -85,B 0,C 180,E1 10334.87,E2 10334.87} C_VEL
LIN {X 0,Y 405.797,Z 616.736,A -85,B 0,C 180,E1 10336.362,E2 10336.362} C_VEL
LIN {X 0,Y 403.025,Z 621.563,A -85,B 0,C 180,E1 10338.05,E2 10338.05} C_VEL
LIN {X 0,Y 397.353,Z 627.355,A -85,B 0,C 180,E1 10340.65,E2 10340.65} C_VEL
LIN {X 0,Y 397.234,Z 627.918,A -85,B 0,C 180,E1 10340.956,E2 10340.956} C_VEL
LIN {X 0,Y 397.028,Z 634.469,A -85,B 0,C 180,E1 10345.623,E2 10345.623} C_VEL
LIN {X 0,Y 397.018,Z 636.517,A -85,B 0,C 180,E1 10349.997,E2 10349.997} C_VEL
LIN {X 0,Y 397.015,Z 634.475,A -85,B 0,C 180,E1 10354.371,E2 10354.371} C_VEL
LIN {X 0,Y 397.258,Z 627.4,A -85,B 0,C 180,E1 10359.318,E2 10359.318} C_VEL
LIN {X 0,Y 398.041,Z 614.596,A -85,B 0,C 180,E1 10364.397,E2 10364.397} C_VEL
LIN {X 0,Y 399.887,Z 596.44,A -85,B 0,C 180,E1 10369.228,E2 10369.228} C_VEL
LIN {X 0,Y 403.127,Z 572.191,A -85,B 0,C 180,E1 10373.864,E2 10373.864} C_VEL
LIN {X 0,Y 407.551,Z 542.722,A -85,B 0,C 180,E1 10377.965,E2 10377.965} C_VEL
LIN {X 0,Y 412.304,Z 510.146,A -85,B 0,C 180,E1 10381.232,E2 10381.232} C_VEL
LIN {X 0,Y 416.743,Z 475.824,A -85,B 0,C 180,E1 10383.656,E2 10383.656} C_VEL
LIN {X 0,Y 420.278,Z 439.102,A -85,B 0,C 180,E1 10385.33,E2 10385.33} C_VEL
LIN {X 0,Y 420.25,Z 428.542,A -85,B 0,C 180,E1 10385.732,E2 10385.732} C_VEL
LIN {X 0,Y 408.216,Z 397.811,A -85,B 0,C 180,E1 10387.668,E2 10387.668} C_VEL
LIN {X 0,Y 395.192,Z 370.16,A -85,B 0,C 180,E1 10389.775,E2 10389.775} C_VEL
LIN {X 0,Y 395.063,Z 370.16,A -85,B 0,C 180,E1 10396.723,E2 10396.723} C_VEL
LIN {X 0,Y 395.13,Z 370.16,A -85,B 0,C 180,E1 10403.567,E2 10403.567} C_VEL
LIN {X 0,Y 395.361,Z 370.456,A -85,B 0,C 180,E1 10407.137,E2 10407.137} C_VEL
LIN {X 0,Y 407.82,Z 397.274,A -85,B 0,C 180,E1 10409.713,E2 10409.713} C_VEL
LIN {X 0,Y 413.821,Z 418.923,A -85,B 0,C 180,E1 10411.153,E2 10411.153} C_VEL
LIN {X 0,Y 411.198,Z 454.782,A -85,B 0,C 180,E1 10413.042,E2 10413.042} C_VEL
LIN {X 0,Y 408.046,Z 486.555,A -85,B 0,C 180,E1 10415.655,E2 10415.655} C_VEL
LIN {X 0,Y 404.714,Z 513.871,A -85,B 0,C 180,E1 10418.91,E2 10418.91} C_VEL
LIN {X 0,Y 401.857,Z 536.381,A -85,B 0,C 180,E1 10422.741,E2 10422.741} C_VEL
LIN {X 0,Y 399.635,Z 553.184,A -85,B 0,C 180,E1 10426.861,E2 10426.861} C_VEL
LIN {X 0,Y 398.204,Z 565.456,A -85,B 0,C 180,E1 10431.591,E2 10431.591} C_VEL
LIN {X 0,Y 397.634,Z 571.131,A -85,B 0,C 180,E1 10435.632,E2 10435.632} C_VEL
LIN {X 0,Y 397.419,Z 572.615,A -85,B 0,C 180,E1 10439.999,E2 10439.999} C_VEL
LIN {X 0,Y 397.416,Z 569.437,A -85,B 0,C 180,E1 10444.368,E2 10444.368} C_VEL
LIN {X 0,Y 397.984,Z 561.43,A -85,B 0,C 180,E1 10448.751,E2 10448.751} C_VEL
LIN {X 0,Y 399.018,Z 547.866,A -85,B 0,C 180,E1 10453.157,E2 10453.157} C_VEL
LIN {X 0,Y 400.932,Z 528.995,A -85,B 0,C 180,E1 10457.297,E2 10457.297} C_VEL
LIN {X 0,Y 403.529,Z 504.577,A -85,B 0,C 180,E1 10461.08,E2 10461.08} C_VEL
LIN {X 0,Y 406.406,Z 476.347,A -85,B 0,C 180,E1 10464.188,E2 10464.188} C_VEL
LIN {X 0,Y 409.219,Z 443.318,A -85,B 0,C 180,E1 10466.688,E2 10466.688} C_VEL
LIN {X 0,Y 410.347,Z 416.624,A -85,B 0,C 180,E1 10468.067,E2 10468.067} C_VEL
LIN {X 0,Y 398.378,Z 379.343,A -85,B 0,C 180,E1 10469.944,E2 10469.944} C_VEL
LIN {X 0,Y 395.531,Z 370.16,A -85,B 0,C 180,E1 10470.353,E2 10470.353} C_VEL
LIN {X 0,Y 395.259,Z 370.16,A -85,B 0,C 180,E1 10477.792,E2 10477.792} C_VEL
LIN {X 0,Y 395.256,Z 370.16,A -85,B 0,C 180,E1 10483.583,E2 10483.583} C_VEL
LIN {X 0,Y 395.23,Z 370.16,A -85,B 0,C 180,E1 10490.002,E2 10490.002} C_VEL
LIN {X 0,Y 395.264,Z 370.245,A -85,B 0,C 180,E1 10495.463,E2 10495.463} C_VEL
LIN {X 0,Y 401.881,Z 384.309,A -85,B 0,C 180,E1 10496.453,E2 10496.453} C_VEL
LIN {X 0,Y 415.758,Z 416.107,A -85,B 0,C 180,E1 10498.884,E2 10498.884} C_VEL
LIN {X 0,Y 419.78,Z 430.43,A -85,B 0,C 180,E1 10499.987,E2 10499.987} C_VEL
LIN {X 0,Y 416.123,Z 461.361,A -85,B 0,C 180,E1 10501.925,E2 10501.925} C_VEL
LIN {X 0,Y 411.48,Z 491.276,A -85,B 0,C 180,E1 10504.73,E2 10504.73} C_VEL
LIN {X 0,Y 406.818,Z 516.546,A -85,B 0,C 180,E1 10508.156,E2 10508.156} C_VEL
LIN {X 0,Y 402.775,Z 537.771,A -85,B 0,C 180,E1 10512.221,E2 10512.221} C_VEL
LIN {X 0,Y 399.769,Z 554.367,A -85,B 0,C 180,E1 10516.87,E2 10516.87} C_VEL
LIN {X 0,Y 398.283,Z 564.587,A -85,B 0,C 180,E1 10521.258,E2 10521.258} C_VEL
LIN {X 0,Y 397.552,Z 570.393,A -85,B 0,C 180,E1 10525.635,E2 10525.635} C_VEL
LIN {X 0,Y 397.317,Z 572.247,A -85,B 0,C 180,E1 10530.003,E2 10530.003} C_VEL
LIN {X 0,Y 397.691,Z 569.183,A -85,B 0,C 180,E1 10535.464,E2 10535.464} C_VEL
LIN {X 0,Y 398.701,Z 561.181,A -85,B 0,C 180,E1 10540.339,E2 10540.339} C_VEL
LIN {X 0,Y 400.988,Z 547.063,A -85,B 0,C 180,E1 10545.328,E2 10545.328} C_VEL
LIN {X 0,Y 404.568,Z 528.234,A -85,B 0,C 180,E1 10549.685,E2 10549.685} C_VEL
LIN {X 0,Y 409.164,Z 504.051,A -85,B 0,C 180,E1 10553.586,E2 10553.586} C_VEL
LIN {X 0,Y 413.806,Z 477.129,A -85,B 0,C 180,E1 10556.63,E2 10556.63} C_VEL
LIN {X 0,Y 418.014,Z 446.258,A -85,B 0,C 180,E1 10559.029,E2 10559.029} C_VEL
LIN {X 0,Y 419.688,Z 428.301,A -85,B 0,C 180,E1 10560.036,E2 10560.036} C_VEL
LIN {X 0,Y 408.175,Z 397.414,A -85,B 0,C 180,E1 10562.46,E2 10562.46} C_VEL
LIN {X 0,Y 395.218,Z 370.16,A -85,B 0,C 180,E1 10564.543,E2 10564.543} C_VEL
LIN {X 0,Y 395.141,Z 370.16,A -85,B 0,C 180,E1 10570.646,E2 10570.646} C_VEL
LIN {X 0,Y 395.196,Z 370.16,A -85,B 0,C 180,E1 10576.712,E2 10576.712} C_VEL
LIN {X 0,Y 395.146,Z 370.16,A -85,B 0,C 180,E1 10583.575,E2 10583.575} C_VEL
LIN {X 0,Y 395.365,Z 370.16,A -85,B 0,C 180,E1 10590.148,E2 10590.148} C_VEL
LIN {X 0,Y 395.622,Z 370.16,A -85,B 0,C 180,E1 10597.503,E2 10597.503} C_VEL
LIN {X 0,Y 395.934,Z 370.16,A -85,B 0,C 180,E1 10604.477,E2 10604.477} C_VEL
LIN {X 0,Y 396.18,Z 370.16,A -85,B 0,C 180,E1 10611.301,E2 10611.301} C_VEL
LIN {X 0,Y 396.492,Z 370.16,A -85,B 0,C 180,E1 10617.813,E2 10617.813} C_VEL
LIN {X 0,Y 396.332,Z 370.16,A -85,B 0,C 180,E1 10624.383,E2 10624.383} C_VEL
LIN {X 0,Y 396.022,Z 370.16,A -85,B 0,C 180,E1 10631.021,E2 10631.021} C_VEL
LIN {X 0,Y 395.794,Z 370.16,A -85,B 0,C 180,E1 10637.82,E2 10637.82} C_VEL
LIN {X 0,Y 395.526,Z 370.16,A -85,B 0,C 180,E1 10644.901,E2 10644.901} C_VEL
LIN {X 0,Y 395.384,Z 370.16,A -85,B 0,C 180,E1 10649.854,E2 10649.854} C_VEL
LIN {X 0,Y 395.214,Z 370.16,A -85,B 0,C 180,E1 10656.438,E2 10656.438} C_VEL
LIN {X 0,Y 395.234,Z 370.16,A -85,B 0,C 180,E1 10663.59,E2 10663.59} C_VEL
LIN {X 0,Y 395.237,Z 370.192,A -85,B 0,C 180,E1 10670.357,E2 10670.357} C_VEL
LIN {X 0,Y 417.16,Z 419.301,A -85,B 0,C 180,E1 10673.701,E2 10673.701} C_VEL
LIN {X 0,Y 420.891,Z 431.472,A -85,B 0,C 180,E1 10674.426,E2 10674.426} C_VEL
LIN {X 0,Y 417.549,Z 467.932,A -85,B 0,C 180,E1 10675.918,E2 10675.918} C_VEL
LIN {X 0,Y 413.419,Z 501.985,A -85,B 0,C 180,E1 10678.114,E2 10678.114} C_VEL
LIN {X 0,Y 408.652,Z 535.448,A -85,B 0,C 180,E1 10681.206,E2 10681.206} C_VEL
LIN {X 0,Y 404.111,Z 565.653,A -85,B 0,C 180,E1 10685.114,E2 10685.114} C_VEL
LIN {X 0,Y 400.656,Z 590.738,A -85,B 0,C 180,E1 10689.538,E2 10689.538} C_VEL
LIN {X 0,Y 398.308,Z 611.174,A -85,B 0,C 180,E1 10694.567,E2 10694.567} C_VEL
LIN {X 0,Y 397.358,Z 625.076,A -85,B 0,C 180,E1 10699.57,E2 10699.57} C_VEL
LIN {X 0,Y 397.234,Z 627.918,A -85,B 0,C 180,E1 10700.956,E2 10700.956} C_VEL
LIN {X 0,Y 395.925,Z 630.021,A -85,B 0,C 180,E1 10702.168,E2 10702.168} C_VEL
LIN {X 0,Y 389.251,Z 633.835,A -85,B 0,C 180,E1 10705.538,E2 10705.538} C_VEL
LIN {X 0,Y 389.125,Z 634.045,A -85,B 0,C 180,E1 10705.861,E2 10705.861} C_VEL
LIN {X 0,Y 389.142,Z 635.88,A -85,B 0,C 180,E1 10709.997,E2 10709.997} C_VEL
LIN {X 0,Y 389.157,Z 633.833,A -85,B 0,C 180,E1 10714.459,E2 10714.459} C_VEL
LIN {X 0,Y 389.389,Z 626.733,A -85,B 0,C 180,E1 10719.508,E2 10719.508} C_VEL
LIN {X 0,Y 390.248,Z 613.621,A -85,B 0,C 180,E1 10724.781,E2 10724.781} C_VEL
LIN {X 0,Y 392.218,Z 595.307,A -85,B 0,C 180,E1 10729.707,E2 10729.707} C_VEL
LIN {X 0,Y 395.676,Z 571.545,A -85,B 0,C 180,E1 10734.316,E2 10734.316} C_VEL
LIN {X 0,Y 400.176,Z 543.039,A -85,B 0,C 180,E1 10738.373,E2 10738.373} C_VEL
LIN {X 0,Y 405.135,Z 510.871,A -85,B 0,C 180,E1 10741.679,E2 10741.679} C_VEL
LIN {X 0,Y 409.731,Z 477.087,A -85,B 0,C 180,E1 10744.133,E2 10744.133} C_VEL
LIN {X 0,Y 413.498,Z 440.793,A -85,B 0,C 180,E1 10745.856,E2 10745.856} C_VEL
LIN {X 0,Y 413.601,Z 430.816,A -85,B 0,C 180,E1 10746.251,E2 10746.251} C_VEL
LIN {X 0,Y 401.634,Z 400.069,A -85,B 0,C 180,E1 10748.274,E2 10748.274} C_VEL
LIN {X 0,Y 387.274,Z 370.16,A -85,B 0,C 180,E1 10750.595,E2 10750.595} C_VEL
LIN {X 0,Y 387.083,Z 370.16,A -85,B 0,C 180,E1 10758.325,E2 10758.325} C_VEL
LIN {X 0,Y 387.34,Z 370.391,A -85,B 0,C 180,E1 10765.797,E2 10765.797} C_VEL
LIN {X 0,Y 390.211,Z 376.194,A -85,B 0,C 180,E1 10766.579,E2 10766.579} C_VEL
LIN {X 0,Y 400.889,Z 398.225,A -85,B 0,C 180,E1 10768.953,E2 10768.953} C_VEL
LIN {X 0,Y 407.227,Z 420.351,A -85,B 0,C 180,E1 10770.568,E2 10770.568} C_VEL
LIN {X 0,Y 404.52,Z 454.842,A -85,B 0,C 180,E1 10772.426,E2 10772.426} C_VEL
LIN {X 0,Y 401.211,Z 486.335,A -85,B 0,C 180,E1 10775.04,E2 10775.04} C_VEL
LIN {X 0,Y 397.755,Z 512.733,A -85,B 0,C 180,E1 10778.169,E2 10778.169} C_VEL
LIN {X 0,Y 394.568,Z 536.089,A -85,B 0,C 180,E1 10782.123,E2 10782.123} C_VEL
LIN {X 0,Y 392.184,Z 552.253,A -85,B 0,C 180,E1 10786.037,E2 10786.037} C_VEL
LIN {X 0,Y 390.656,Z 564.561,A -85,B 0,C 180,E1 10790.519,E2 10790.519} C_VEL
LIN {X 0,Y 389.786,Z 571.914,A -85,B 0,C 180,E1 10795.543,E2 10795.543} C_VEL
LIN {X 0,Y 389.546,Z 573.287,A -85,B 0,C 180,E1 10799.999,E2 10799.999} C_VEL
LIN {X 0,Y 389.577,Z 569.976,A -85,B 0,C 180,E1 10804.456,E2 10804.456} C_VEL
LIN {X 0,Y 390.155,Z 561.79,A -85,B 0,C 180,E1 10808.928,E2 10808.928} C_VEL
LIN {X 0,Y 391.246,Z 548.039,A -85,B 0,C 180,E1 10813.423,E2 10813.423} C_VEL
LIN {X 0,Y 393.274,Z 528.862,A -85,B 0,C 180,E1 10817.645,E2 10817.645} C_VEL
LIN {X 0,Y 395.981,Z 504.467,A -85,B 0,C 180,E1 10821.442,E2 10821.442} C_VEL
LIN {X 0,Y 399.044,Z 475.229,A -85,B 0,C 180,E1 10824.664,E2 10824.664} C_VEL
LIN {X 0,Y 401.918,Z 442.364,A -85,B 0,C 180,E1 10827.144,E2 10827.144} C_VEL
LIN {X 0,Y 403.005,Z 418.473,A -85,B 0,C 180,E1 10828.401,E2 10828.401} C_VEL
LIN {X 0,Y 391.344,Z 381.852,A -85,B 0,C 180,E1 10830.328,E2 10830.328} C_VEL
LIN {X 0,Y 387.551,Z 370.16,A -85,B 0,C 180,E1 10830.981,E2 10830.981} C_VEL
LIN {X 0,Y 387.345,Z 370.16,A -85,B 0,C 180,E1 10835.89,E2 10835.89} C_VEL
LIN {X 0,Y 387.244,Z 370.16,A -85,B 0,C 180,E1 10842.034,E2 10842.034} C_VEL
LIN {X 0,Y 387.232,Z 370.16,A -85,B 0,C 180,E1 10848.35,E2 10848.35} C_VEL
LIN {X 0,Y 387.333,Z 370.831,A -85,B 0,C 180,E1 10854.582,E2 10854.582} C_VEL
LIN {X 0,Y 405.269,Z 408.6,A -85,B 0,C 180,E1 10857.546,E2 10857.546} C_VEL
LIN {X 0,Y 413.087,Z 431.212,A -85,B 0,C 180,E1 10859.422,E2 10859.422} C_VEL
LIN {X 0,Y 409.222,Z 462.298,A -85,B 0,C 180,E1 10861.408,E2 10861.408} C_VEL
LIN {X 0,Y 404.54,Z 491.355,A -85,B 0,C 180,E1 10864.174,E2 10864.174} C_VEL
LIN {X 0,Y 399.502,Z 517.277,A -85,B 0,C 180,E1 10867.735,E2 10867.735} C_VEL
LIN {X 0,Y 395.271,Z 538.453,A -85,B 0,C 180,E1 10871.872,E2 10871.872} C_VEL
LIN {X 0,Y 392.059,Z 555.031,A -85,B 0,C 180,E1 10876.607,E2 10876.607} C_VEL
LIN {X 0,Y 390.384,Z 565.831,A -85,B 0,C 180,E1 10881.443,E2 10881.443} C_VEL
LIN {X 0,Y 389.707,Z 571.031,A -85,B 0,C 180,E1 10885.547,E2 10885.547} C_VEL
LIN {X 0,Y 389.442,Z 572.884,A -85,B 0,C 180,E1 10890.003,E2 10890.003} C_VEL
LIN {X 0,Y 389.85,Z 569.823,A -85,B 0,C 180,E1 10895.575,E2 10895.575} C_VEL
LIN {X 0,Y 390.932,Z 561.714,A -85,B 0,C 180,E1 10900.603,E2 10900.603} C_VEL
LIN {X 0,Y 393.354,Z 547.739,A -85,B 0,C 180,E1 10905.633,E2 10905.633} C_VEL
LIN {X 0,Y 397.138,Z 528.943,A -85,B 0,C 180,E1 10910.069,E2 10910.069} C_VEL
LIN {X 0,Y 401.772,Z 505.841,A -85,B 0,C 180,E1 10913.899,E2 10913.899} C_VEL
LIN {X 0,Y 406.808,Z 477.988,A -85,B 0,C 180,E1 10917.125,E2 10917.125} C_VEL
LIN {X 0,Y 411.204,Z 447.342,A -85,B 0,C 180,E1 10919.557,E2 10919.557} C_VEL
LIN {X 0,Y 412.593,Z 429.749,A -85,B 0,C 180,E1 10920.604,E2 10920.604} C_VEL
LIN {X 0,Y 400.9,Z 398.454,A -85,B 0,C 180,E1 10923.165,E2 10923.165} C_VEL
LIN {X 0,Y 387.375,Z 371.509,A -85,B 0,C 180,E1 10925.292,E2 10925.292} C_VEL
LIN {X 0,Y 387.245,Z 370.16,A -85,B 0,C 180,E1 10925.412,E2 10925.412} C_VEL
LIN {X 0,Y 387.144,Z 370.16,A -85,B 0,C 180,E1 10932.016,E2 10932.016} C_VEL
LIN {X 0,Y 387.198,Z 370.16,A -85,B 0,C 180,E1 10938.344,E2 10938.344} C_VEL
LIN {X 0,Y 387.277,Z 370.16,A -85,B 0,C 180,E1 10945.183,E2 10945.183} C_VEL
LIN {X 0,Y 387.5,Z 370.16,A -85,B 0,C 180,E1 10952.044,E2 10952.044} C_VEL
LIN {X 0,Y 387.817,Z 370.16,A -85,B 0,C 180,E1 10959.546,E2 10959.546} C_VEL
LIN {X 0,Y 388.096,Z 370.16,A -85,B 0,C 180,E1 10966.466,E2 10966.466} C_VEL
LIN {X 0,Y 388.383,Z 370.16,A -85,B 0,C 180,E1 10973.286,E2 10973.286} C_VEL
LIN {X 0,Y 388.725,Z 370.16,A -85,B 0,C 180,E1 10980.001,E2 10980.001} C_VEL
LIN {X 0,Y 388.412,Z 370.16,A -85,B 0,C 180,E1 10986.716,E2 10986.716} C_VEL
LIN {X 0,Y 388.03,Z 370.16,A -85,B 0,C 180,E1 10993.54,E2 10993.54} C_VEL
LIN {X 0,Y 387.792,Z 370.16,A -85,B 0,C 180,E1 11000.572,E2 11000.572} C_VEL
LIN {X 0,Y 387.512,Z 370.16,A -85,B 0,C 180,E1 11007.959,E2 11007.959} C_VEL
LIN {X 0,Y 387.302,Z 370.16,A -85,B 0,C 180,E1 11015.899,E2 11015.899} C_VEL
LIN {X 0,Y 387.226,Z 370.16,A -85,B 0,C 180,E1 11022.021,E2 11022.021} C_VEL
LIN {X 0,Y 387.341,Z 370.25,A -85,B 0,C 180,E1 11029.476,E2 11029.476} C_VEL
LIN {X 0,Y 393.921,Z 384.483,A -85,B 0,C 180,E1 11030.557,E2 11030.557} C_VEL
LIN {X 0,Y 410.743,Z 422.25,A -85,B 0,C 180,E1 11033.205,E2 11033.205} C_VEL
LIN {X 0,Y 414.038,Z 433.84,A -85,B 0,C 180,E1 11033.917,E2 11033.917} C_VEL
LIN {X 0,Y 410.556,Z 469.775,A -85,B 0,C 180,E1 11035.458,E2 11035.458} C_VEL
LIN {X 0,Y 405.994,Z 505.178,A -85,B 0,C 180,E1 11037.842,E2 11037.842} C_VEL
LIN {X 0,Y 400.948,Z 538.162,A -85,B 0,C 180,E1 11041.063,E2 11041.063} C_VEL
LIN {X 0,Y 396.409,Z 566.673,A -85,B 0,C 180,E1 11044.899,E2 11044.899} C_VEL
LIN {X 0,Y 392.849,Z 591.32,A -85,B 0,C 180,E1 11049.408,E2 11049.408} C_VEL
LIN {X 0,Y 390.529,Z 610.462,A -85,B 0,C 180,E1 11054.251,E2 11054.251} C_VEL
LIN {X 0,Y 389.488,Z 624.397,A -85,B 0,C 180,E1 11059.357,E2 11059.357} C_VEL
LIN {X 0,Y 389.188,Z 632.694,A -85,B 0,C 180,E1 11064.416,E2 11064.416} C_VEL
LIN {X 0,Y 389.125,Z 634.045,A -85,B 0,C 180,E1 11065.861,E2 11065.861} C_VEL
LIN {X 0,Y 387.795,Z 634.899,A -85,B 0,C 180,E1 11067.128,E2 11067.128} C_VEL
LIN {X 0,Y 381.284,Z 635.155,A -85,B 0,C 180,E1 11070.606,E2 11070.606} C_VEL
LIN {X 0,Y 381.185,Z 635.014,A -85,B 0,C 180,E1 11070.936,E2 11070.936} C_VEL
LIN {X 0,Y 381.3,Z 632.056,A -85,B 0,C 180,E1 11075.693,E2 11075.693} C_VEL
LIN {X 0,Y 381.625,Z 623.738,A -85,B 0,C 180,E1 11080.858,E2 11080.858} C_VEL
LIN {X 0,Y 382.792,Z 609.79,A -85,B 0,C 180,E1 11086.069,E2 11086.069} C_VEL
LIN {X 0,Y 385.416,Z 589.266,A -85,B 0,C 180,E1 11091.302,E2 11091.302} C_VEL
LIN {X 0,Y 389.426,Z 563.746,A -85,B 0,C 180,E1 11095.946,E2 11095.946} C_VEL
LIN {X 0,Y 394.404,Z 533.758,A -85,B 0,C 180,E1 11099.931,E2 11099.931} C_VEL
LIN {X 0,Y 399.497,Z 501.211,A -85,B 0,C 180,E1 11103.024,E2 11103.024} C_VEL
LIN {X 0,Y 404.31,Z 465.504,A -85,B 0,C 180,E1 11105.364,E2 11105.364} C_VEL
LIN {X 0,Y 406.947,Z 433.138,A -85,B 0,C 180,E1 11106.772,E2 11106.772} C_VEL
LIN {X 0,Y 395.852,Z 404.129,A -85,B 0,C 180,E1 11108.778,E2 11108.778} C_VEL
LIN {X 0,Y 379.351,Z 371.488,A -85,B 0,C 180,E1 11111.448,E2 11111.448} C_VEL
LIN {X 0,Y 379.247,Z 370.16,A -85,B 0,C 180,E1 11111.582,E2 11111.582} C_VEL
LIN {X 0,Y 379.105,Z 370.16,A -85,B 0,C 180,E1 11119.349,E2 11119.349} C_VEL
LIN {X 0,Y 379.379,Z 370.843,A -85,B 0,C 180,E1 11124.186,E2 11124.186} C_VEL
LIN {X 0,Y 382.257,Z 376.234,A -85,B 0,C 180,E1 11125.134,E2 11125.134} C_VEL
LIN {X 0,Y 391.295,Z 393.214,A -85,B 0,C 180,E1 11127.497,E2 11127.497} C_VEL
LIN {X 0,Y 399.219,Z 414.699,A -85,B 0,C 180,E1 11129.418,E2 11129.418} C_VEL
LIN {X 0,Y 400.588,Z 425.872,A -85,B 0,C 180,E1 11130.133,E2 11130.133} C_VEL
LIN {X 0,Y 397.413,Z 460.733,A -85,B 0,C 180,E1 11132.181,E2 11132.181} C_VEL
LIN {X 0,Y 393.714,Z 491.894,A -85,B 0,C 180,E1 11134.976,E2 11134.976} C_VEL
LIN {X 0,Y 389.69,Z 519.563,A -85,B 0,C 180,E1 11138.567,E2 11138.567} C_VEL
LIN {X 0,Y 386.524,Z 541.147,A -85,B 0,C 180,E1 11142.622,E2 11142.622} C_VEL
LIN {X 0,Y 384.049,Z 556.869,A -85,B 0,C 180,E1 11146.898,E2 11146.898} C_VEL
LIN {X 0,Y 382.56,Z 567.864,A -85,B 0,C 180,E1 11151.604,E2 11151.604} C_VEL
LIN {X 0,Y 381.973,Z 572.716,A -85,B 0,C 180,E1 11155.452,E2 11155.452} C_VEL
LIN {X 0,Y 381.697,Z 573.956,A -85,B 0,C 180,E1 11159.999,E2 11159.999} C_VEL
LIN {X 0,Y 381.708,Z 570.518,A -85,B 0,C 180,E1 11164.548,E2 11164.548} C_VEL
LIN {X 0,Y 382.331,Z 562.133,A -85,B 0,C 180,E1 11169.112,E2 11169.112} C_VEL
LIN {X 0,Y 383.478,Z 548.179,A -85,B 0,C 180,E1 11173.7,E2 11173.7} C_VEL
LIN {X 0,Y 385.634,Z 528.688,A -85,B 0,C 180,E1 11178.007,E2 11178.007} C_VEL
LIN {X 0,Y 388.505,Z 503.899,A -85,B 0,C 180,E1 11181.876,E2 11181.876} C_VEL
LIN {X 0,Y 391.668,Z 474.096,A -85,B 0,C 180,E1 11185.16,E2 11185.16} C_VEL
LIN {X 0,Y 394.711,Z 440.739,A -85,B 0,C 180,E1 11187.656,E2 11187.656} C_VEL
LIN {X 0,Y 395.416,Z 419.469,A -85,B 0,C 180,E1 11188.802,E2 11188.802} C_VEL
LIN {X 0,Y 384.293,Z 384.371,A -85,B 0,C 180,E1 11190.711,E2 11190.711} C_VEL
LIN {X 0,Y 379.601,Z 370.16,A -85,B 0,C 180,E1 11191.457,E2 11191.457} C_VEL
LIN {X 0,Y 379.325,Z 370.16,A -85,B 0,C 180,E1 11197.045,E2 11197.045} C_VEL
LIN {X 0,Y 379.264,Z 370.16,A -85,B 0,C 180,E1 11204.073,E2 11204.073} C_VEL
LIN {X 0,Y 379.246,Z 370.16,A -85,B 0,C 180,E1 11210.309,E2 11210.309} C_VEL
LIN {X 0,Y 379.321,Z 370.347,A -85,B 0,C 180,E1 11213.62,E2 11213.62} C_VEL
LIN {X 0,Y 384.159,Z 380.536,A -85,B 0,C 180,E1 11214.418,E2 11214.418} C_VEL
LIN {X 0,Y 399.113,Z 412.339,A -85,B 0,C 180,E1 11217.071,E2 11217.071} C_VEL
LIN {X 0,Y 406.199,Z 434.072,A -85,B 0,C 180,E1 11218.954,E2 11218.954} C_VEL
LIN {X 0,Y 402.114,Z 464.9,A -85,B 0,C 180,E1 11221.009,E2 11221.009} C_VEL
LIN {X 0,Y 397.071,Z 494.07,A -85,B 0,C 180,E1 11223.91,E2 11223.91} C_VEL
LIN {X 0,Y 391.804,Z 520.021,A -85,B 0,C 180,E1 11227.632,E2 11227.632} C_VEL
LIN {X 0,Y 387.256,Z 541.417,A -85,B 0,C 180,E1 11232.073,E2 11232.073} C_VEL
LIN {X 0,Y 384.058,Z 557.231,A -85,B 0,C 180,E1 11236.903,E2 11236.903} C_VEL
LIN {X 0,Y 382.321,Z 567.927,A -85,B 0,C 180,E1 11242.19,E2 11242.19} C_VEL
LIN {X 0,Y 381.866,Z 571.668,A -85,B 0,C 180,E1 11245.456,E2 11245.456} C_VEL
LIN {X 0,Y 381.567,Z 573.521,A -85,B 0,C 180,E1 11250.003,E2 11250.003} C_VEL
LIN {X 0,Y 381.994,Z 570.465,A -85,B 0,C 180,E1 11255.69,E2 11255.69} C_VEL
LIN {X 0,Y 383.182,Z 562.367,A -85,B 0,C 180,E1 11260.82,E2 11260.82} C_VEL
LIN {X 0,Y 385.741,Z 548.41,A -85,B 0,C 180,E1 11265.949,E2 11265.949} C_VEL
LIN {X 0,Y 389.722,Z 529.649,A -85,B 0,C 180,E1 11270.467,E2 11270.467} C_VEL
LIN {X 0,Y 394.799,Z 505.595,A -85,B 0,C 180,E1 11274.499,E2 11274.499} C_VEL
LIN {X 0,Y 400.062,Z 477.487,A -85,B 0,C 180,E1 11277.774,E2 11277.774} C_VEL
LIN {X 0,Y 404.643,Z 446.326,A -85,B 0,C 180,E1 11280.239,E2 11280.239} C_VEL
LIN {X 0,Y 405.635,Z 431.45,A -85,B 0,C 180,E1 11281.167,E2 11281.167} C_VEL
LIN {X 0,Y 393.751,Z 399.77,A -85,B 0,C 180,E1 11283.879,E2 11283.879} C_VEL
LIN {X 0,Y 379.351,Z 371.158,A -85,B 0,C 180,E1 11286.25,E2 11286.25} C_VEL
LIN {X 0,Y 379.243,Z 370.16,A -85,B 0,C 180,E1 11286.472,E2 11286.472} C_VEL
LIN {X 0,Y 379.18,Z 370.16,A -85,B 0,C 180,E1 11294.058,E2 11294.058} C_VEL
LIN {X 0,Y 379.202,Z 370.16,A -85,B 0,C 180,E1 11300.301,E2 11300.301} C_VEL
LIN {X 0,Y 379.397,Z 370.16,A -85,B 0,C 180,E1 11306.933,E2 11306.933} C_VEL
LIN {X 0,Y 379.625,Z 370.16,A -85,B 0,C 180,E1 11313.983,E2 11313.983} C_VEL
LIN {X 0,Y 379.963,Z 370.16,A -85,B 0,C 180,E1 11321.414,E2 11321.414} C_VEL
LIN {X 0,Y 380.256,Z 370.16,A -85,B 0,C 180,E1 11328.519,E2 11328.519} C_VEL
LIN {X 0,Y 380.606,Z 370.16,A -85,B 0,C 180,E1 11335.439,E2 11335.439} C_VEL
LIN {X 0,Y 380.791,Z 370.16,A -85,B 0,C 180,E1 11342.28,E2 11342.28} C_VEL
LIN {X 0,Y 380.313,Z 370.16,A -85,B 0,C 180,E1 11349.164,E2 11349.164} C_VEL
LIN {X 0,Y 379.99,Z 370.16,A -85,B 0,C 180,E1 11356.195,E2 11356.195} C_VEL
LIN {X 0,Y 379.678,Z 370.16,A -85,B 0,C 180,E1 11363.501,E2 11363.501} C_VEL
LIN {X 0,Y 379.413,Z 370.16,A -85,B 0,C 180,E1 11371.248,E2 11371.248} C_VEL
LIN {X 0,Y 379.293,Z 370.16,A -85,B 0,C 180,E1 11377.027,E2 11377.027} C_VEL
LIN {X 0,Y 379.246,Z 370.16,A -85,B 0,C 180,E1 11384.06,E2 11384.06} C_VEL
LIN {X 0,Y 379.389,Z 370.893,A -85,B 0,C 180,E1 11388.556,E2 11388.556} C_VEL
LIN {X 0,Y 402.058,Z 418.889,A -85,B 0,C 180,E1 11392.256,E2 11392.256} C_VEL
LIN {X 0,Y 407.218,Z 436.322,A -85,B 0,C 180,E1 11393.394,E2 11393.394} C_VEL
LIN {X 0,Y 403.347,Z 473.342,A -85,B 0,C 180,E1 11395.073,E2 11395.073} C_VEL
LIN {X 0,Y 398.416,Z 508.774,A -85,B 0,C 180,E1 11397.615,E2 11397.615} C_VEL
LIN {X 0,Y 393.282,Z 540.882,A -85,B 0,C 180,E1 11400.918,E2 11400.918} C_VEL
LIN {X 0,Y 388.466,Z 569.194,A -85,B 0,C 180,E1 11404.92,E2 11404.92} C_VEL
LIN {X 0,Y 384.79,Z 592.973,A -85,B 0,C 180,E1 11409.524,E2 11409.524} C_VEL
LIN {X 0,Y 382.551,Z 611.614,A -85,B 0,C 180,E1 11414.503,E2 11414.503} C_VEL
LIN {X 0,Y 381.561,Z 624.96,A -85,B 0,C 180,E1 11419.711,E2 11419.711} C_VEL
LIN {X 0,Y 381.327,Z 632.047,A -85,B 0,C 180,E1 11424.3,E2 11424.3} C_VEL
LIN {X 0,Y 381.23,Z 634.684,A -85,B 0,C 180,E1 11427.721,E2 11427.721} C_VEL
LIN {X 0,Y 381.185,Z 635.014,A -85,B 0,C 180,E1 11430.936,E2 11430.936} C_VEL
LIN {X 0,Y 378.705,Z 634.23,A -85,B 0,C 180,E1 11432.87,E2 11432.87} C_VEL
LIN {X 0,Y 373.424,Z 631.085,A -85,B 0,C 180,E1 11436.096,E2 11436.096} C_VEL
LIN {X 0,Y 373.811,Z 621.825,A -85,B 0,C 180,E1 11441.68,E2 11441.68} C_VEL
LIN {X 0,Y 375.294,Z 607.21,A -85,B 0,C 180,E1 11447.002,E2 11447.002} C_VEL
LIN {X 0,Y 378.135,Z 586.524,A -85,B 0,C 180,E1 11452.173,E2 11452.173} C_VEL
LIN {X 0,Y 382.403,Z 561.174,A -85,B 0,C 180,E1 11456.767,E2 11456.767} C_VEL
LIN {X 0,Y 387.547,Z 531.941,A -85,B 0,C 180,E1 11460.632,E2 11460.632} C_VEL
LIN {X 0,Y 392.831,Z 499.228,A -85,B 0,C 180,E1 11463.751,E2 11463.751} C_VEL
LIN {X 0,Y 397.885,Z 463.195,A -85,B 0,C 180,E1 11466.096,E2 11466.096} C_VEL
LIN {X 0,Y 400.207,Z 435.224,A -85,B 0,C 180,E1 11467.33,E2 11467.33} C_VEL
LIN {X 0,Y 389.047,Z 406.011,A -85,B 0,C 180,E1 11469.466,E2 11469.466} C_VEL
LIN {X 0,Y 371.342,Z 371.251,A -85,B 0,C 180,E1 11472.454,E2 11472.454} C_VEL
LIN {X 0,Y 371.216,Z 370.16,A -85,B 0,C 180,E1 11472.768,E2 11472.768} C_VEL
LIN {X 0,Y 371.224,Z 370.16,A -85,B 0,C 180,E1 11479.267,E2 11479.267} C_VEL
LIN {X 0,Y 371.213,Z 370.956,A -85,B 0,C 180,E1 11481.913,E2 11481.913} C_VEL
LIN {X 0,Y 374.453,Z 376.428,A -85,B 0,C 180,E1 11483.343,E2 11483.343} C_VEL
LIN {X 0,Y 381.972,Z 389.114,A -85,B 0,C 180,E1 11485.777,E2 11485.777} C_VEL
LIN {X 0,Y 390.813,Z 409.323,A -85,B 0,C 180,E1 11488.105,E2 11488.105} C_VEL
LIN {X 0,Y 394.347,Z 426.609,A -85,B 0,C 180,E1 11489.444,E2 11489.444} C_VEL
LIN {X 0,Y 390.876,Z 461.514,A -85,B 0,C 180,E1 11491.542,E2 11491.542} C_VEL
LIN {X 0,Y 386.744,Z 493.615,A -85,B 0,C 180,E1 11494.493,E2 11494.493} C_VEL
LIN {X 0,Y 382.549,Z 520.326,A -85,B 0,C 180,E1 11498.047,E2 11498.047} C_VEL
LIN {X 0,Y 379.056,Z 542.31,A -85,B 0,C 180,E1 11502.268,E2 11502.268} C_VEL
LIN {X 0,Y 376.388,Z 557.901,A -85,B 0,C 180,E1 11506.626,E2 11506.626} C_VEL
LIN {X 0,Y 374.758,Z 568.868,A -85,B 0,C 180,E1 11511.489,E2 11511.489} C_VEL
LIN {X 0,Y 374.156,Z 573.509,A -85,B 0,C 180,E1 11515.357,E2 11515.357} C_VEL
LIN {X 0,Y 373.824,Z 574.625,A -85,B 0,C 180,E1 11519.998,E2 11519.998} C_VEL
LIN {X 0,Y 373.865,Z 571.049,A -85,B 0,C 180,E1 11524.644,E2 11524.644} C_VEL
LIN {X 0,Y 374.494,Z 562.463,A -85,B 0,C 180,E1 11529.304,E2 11529.304} C_VEL
LIN {X 0,Y 375.724,Z 548.301,A -85,B 0,C 180,E1 11533.989,E2 11533.989} C_VEL
LIN {X 0,Y 378.02,Z 528.52,A -85,B 0,C 180,E1 11538.382,E2 11538.382} C_VEL
LIN {X 0,Y 380.983,Z 503.312,A -85,B 0,C 180,E1 11542.331,E2 11542.331} C_VEL
LIN {X 0,Y 384.175,Z 474.611,A -85,B 0,C 180,E1 11545.518,E2 11545.518} C_VEL
LIN {X 0,Y 387.345,Z 441.242,A -85,B 0,C 180,E1 11548.055,E2 11548.055} C_VEL
LIN {X 0,Y 387.963,Z 420.884,A -85,B 0,C 180,E1 11549.183,E2 11549.183} C_VEL
LIN {X 0,Y 376.12,Z 383.745,A -85,B 0,C 180,E1 11551.259,E2 11551.259} C_VEL
LIN {X 0,Y 371.657,Z 370.16,A -85,B 0,C 180,E1 11551.973,E2 11551.973} C_VEL
LIN {X 0,Y 371.341,Z 370.16,A -85,B 0,C 180,E1 11559.235,E2 11559.235} C_VEL
LIN {X 0,Y 371.351,Z 370.16,A -85,B 0,C 180,E1 11566.132,E2 11566.132} C_VEL
LIN {X 0,Y 371.387,Z 370.954,A -85,B 0,C 180,E1 11572.637,E2 11572.637} C_VEL
LIN {X 0,Y 389.956,Z 408.497,A -85,B 0,C 180,E1 11575.933,E2 11575.933} C_VEL
LIN {X 0,Y 399.43,Z 435.83,A -85,B 0,C 180,E1 11578.407,E2 11578.407} C_VEL
LIN {X 0,Y 394.987,Z 467.503,A -85,B 0,C 180,E1 11580.592,E2 11580.592} C_VEL
LIN {X 0,Y 389.708,Z 496.412,A -85,B 0,C 180,E1 11583.597,E2 11583.597} C_VEL
LIN {X 0,Y 384.274,Z 521.786,A -85,B 0,C 180,E1 11587.371,E2 11587.371} C_VEL
LIN {X 0,Y 379.741,Z 542.097,A -85,B 0,C 180,E1 11591.706,E2 11591.706} C_VEL
LIN {X 0,Y 376.374,Z 557.884,A -85,B 0,C 180,E1 11596.631,E2 11596.631} C_VEL
LIN {X 0,Y 374.616,Z 567.883,A -85,B 0,C 180,E1 11601.578,E2 11601.578} C_VEL
LIN {X 0,Y 374.015,Z 572.306,A -85,B 0,C 180,E1 11605.36,E2 11605.36} C_VEL
LIN {X 0,Y 373.698,Z 574.158,A -85,B 0,C 180,E1 11610.003,E2 11610.003} C_VEL
LIN {X 0,Y 374.167,Z 571.104,A -85,B 0,C 180,E1 11615.809,E2 11615.809} C_VEL
LIN {X 0,Y 375.405,Z 563.022,A -85,B 0,C 180,E1 11621.047,E2 11621.047} C_VEL
LIN {X 0,Y 378.144,Z 549.079,A -85,B 0,C 180,E1 11626.279,E2 11626.279} C_VEL
LIN {X 0,Y 382.304,Z 530.355,A -85,B 0,C 180,E1 11630.883,E2 11630.883} C_VEL
LIN {X 0,Y 387.632,Z 506.363,A -85,B 0,C 180,E1 11634.983,E2 11634.983} C_VEL
LIN {X 0,Y 393.129,Z 478.336,A -85,B 0,C 180,E1 11638.308,E2 11638.308} C_VEL
LIN {X 0,Y 397.913,Z 447.395,A -85,B 0,C 180,E1 11640.806,E2 11640.806} C_VEL
LIN {X 0,Y 398.885,Z 434.052,A -85,B 0,C 180,E1 11641.663,E2 11641.663} C_VEL
LIN {X 0,Y 387.18,Z 402.145,A -85,B 0,C 180,E1 11644.524,E2 11644.524} C_VEL
LIN {X 0,Y 371.389,Z 371.515,A -85,B 0,C 180,E1 11647.239,E2 11647.239} C_VEL
LIN {X 0,Y 371.248,Z 370.16,A -85,B 0,C 180,E1 11647.428,E2 11647.428} C_VEL
LIN {X 0,Y 371.269,Z 370.16,A -85,B 0,C 180,E1 11653.89,E2 11653.89} C_VEL
LIN {X 0,Y 371.272,Z 370.16,A -85,B 0,C 180,E1 11660.789,E2 11660.789} C_VEL
LIN {X 0,Y 371.456,Z 370.16,A -85,B 0,C 180,E1 11668.008,E2 11668.008} C_VEL
LIN {X 0,Y 371.728,Z 370.16,A -85,B 0,C 180,E1 11675.969,E2 11675.969} C_VEL
LIN {X 0,Y 372.147,Z 370.16,A -85,B 0,C 180,E1 11683.457,E2 11683.457} C_VEL
LIN {X 0,Y 372.408,Z 370.16,A -85,B 0,C 180,E1 11690.643,E2 11690.643} C_VEL
LIN {X 0,Y 372.796,Z 370.16,A -85,B 0,C 180,E1 11697.674,E2 11697.674} C_VEL
LIN {X 0,Y 372.875,Z 370.16,A -85,B 0,C 180,E1 11702.328,E2 11702.328} C_VEL
LIN {X 0,Y 372.374,Z 370.16,A -85,B 0,C 180,E1 11709.361,E2 11709.361} C_VEL
LIN {X 0,Y 372.076,Z 370.16,A -85,B 0,C 180,E1 11716.549,E2 11716.549} C_VEL
LIN {X 0,Y 371.836,Z 370.16,A -85,B 0,C 180,E1 11721.497,E2 11721.497} C_VEL
LIN {X 0,Y 371.634,Z 370.16,A -85,B 0,C 180,E1 11726.624,E2 11726.624} C_VEL
LIN {X 0,Y 371.489,Z 370.16,A -85,B 0,C 180,E1 11731.992,E2 11731.992} C_VEL
LIN {X 0,Y 371.322,Z 370.16,A -85,B 0,C 180,E1 11739.221,E2 11739.221} C_VEL
LIN {X 0,Y 371.337,Z 370.16,A -85,B 0,C 180,E1 11746.12,E2 11746.12} C_VEL
LIN {X 0,Y 371.39,Z 370.454,A -85,B 0,C 180,E1 11747.547,E2 11747.547} C_VEL
LIN {X 0,Y 394.45,Z 418.731,A -85,B 0,C 180,E1 11751.477,E2 11751.477} C_VEL
LIN {X 0,Y 400.584,Z 436.955,A -85,B 0,C 180,E1 11752.79,E2 11752.79} C_VEL
LIN {X 0,Y 396.599,Z 473.464,A -85,B 0,C 180,E1 11754.482,E2 11754.482} C_VEL
LIN {X 0,Y 391.539,Z 508.11,A -85,B 0,C 180,E1 11757.006,E2 11757.006} C_VEL
LIN {X 0,Y 386.12,Z 540.014,A -85,B 0,C 180,E1 11760.326,E2 11760.326} C_VEL
LIN {X 0,Y 381.11,Z 568.42,A -85,B 0,C 180,E1 11764.402,E2 11764.402} C_VEL
LIN {X 0,Y 377.192,Z 592.392,A -85,B 0,C 180,E1 11769.128,E2 11769.128} C_VEL
LIN {X 0,Y 374.765,Z 610.913,A -85,B 0,C 180,E1 11774.173,E2 11774.173} C_VEL
LIN {X 0,Y 373.705,Z 624.291,A -85,B 0,C 180,E1 11779.493,E2 11779.493} C_VEL
LIN {X 0,Y 373.465,Z 631.502,A -85,B 0,C 180,E1 11784.27,E2 11784.27} C_VEL
LIN {X 0,Y 373.416,Z 634.607,A -85,B 0,C 180,E1 11789.997,E2 11789.997} C_VEL
LIN {X 0,Y 373.439,Z 631.533,A -85,B 0,C 180,E1 11795.705,E2 11795.705} C_VEL
LIN {X 0,Y 373.424,Z 631.085,A -85,B 0,C 180,E1 11796.096,E2 11796.096} C_VEL
LIN {X 0,Y 370.96,Z 628.443,A -85,B 0,C 180,E1 11798.042,E2 11798.042} C_VEL
LIN {X 0,Y 365.922,Z 623.243,A -85,B 0,C 180,E1 11800.927,E2 11800.927} C_VEL
LIN {X 0,Y 365.868,Z 622.554,A -85,B 0,C 180,E1 11801.257,E2 11801.257} C_VEL
LIN {X 0,Y 367.262,Z 608.399,A -85,B 0,C 180,E1 11806.768,E2 11806.768} C_VEL
LIN {X 0,Y 370.183,Z 588.382,A -85,B 0,C 180,E1 11812.09,E2 11812.09} C_VEL
LIN {X 0,Y 374.675,Z 562.816,A -85,B 0,C 180,E1 11816.935,E2 11816.935} C_VEL
LIN {X 0,Y 380.181,Z 533.298,A -85,B 0,C 180,E1 11821.006,E2 11821.006} C_VEL
LIN {X 0,Y 385.884,Z 499.623,A -85,B 0,C 180,E1 11824.307,E2 11824.307} C_VEL
LIN {X 0,Y 391.183,Z 463.749,A -85,B 0,C 180,E1 11826.693,E2 11826.693} C_VEL
LIN {X 0,Y 393.459,Z 437.053,A -85,B 0,C 180,E1 11827.925,E2 11827.925} C_VEL
LIN {X 0,Y 381.847,Z 406.985,A -85,B 0,C 180,E1 11830.254,E2 11830.254} C_VEL
LIN {X 0,Y 364.113,Z 373.643,A -85,B 0,C 180,E1 11833.378,E2 11833.378} C_VEL
LIN {X 0,Y 363.296,Z 370.249,A -85,B 0,C 180,E1 11836.469,E2 11836.469} C_VEL
LIN {X 0,Y 366.614,Z 376.589,A -85,B 0,C 180,E1 11840.719,E2 11840.719} C_VEL
LIN {X 0,Y 368.271,Z 378.689,A -85,B 0,C 180,E1 11841.62,E2 11841.62} C_VEL
LIN {X 0,Y 373.391,Z 387.291,A -85,B 0,C 180,E1 11843.843,E2 11843.843} C_VEL
LIN {X 0,Y 380.608,Z 401.078,A -85,B 0,C 180,E1 11846.14,E2 11846.14} C_VEL
LIN {X 0,Y 387.486,Z 421.578,A -85,B 0,C 180,E1 11848.262,E2 11848.262} C_VEL
LIN {X 0,Y 387.925,Z 431.626,A -85,B 0,C 180,E1 11848.922,E2 11848.922} C_VEL
LIN {X 0,Y 384.098,Z 465.638,A -85,B 0,C 180,E1 11851.128,E2 11851.128} C_VEL
LIN {X 0,Y 379.831,Z 495.466,A -85,B 0,C 180,E1 11853.995,E2 11853.995} C_VEL
LIN {X 0,Y 375.292,Z 522.304,A -85,B 0,C 180,E1 11857.685,E2 11857.685} C_VEL
LIN {X 0,Y 371.64,Z 543.584,A -85,B 0,C 180,E1 11861.902,E2 11861.902} C_VEL
LIN {X 0,Y 368.756,Z 558.981,A -85,B 0,C 180,E1 11866.344,E2 11866.344} C_VEL
LIN {X 0,Y 367.209,Z 568.434,A -85,B 0,C 180,E1 11870.506,E2 11870.506} C_VEL
LIN {X 0,Y 366.341,Z 574.318,A -85,B 0,C 180,E1 11875.258,E2 11875.258} C_VEL
LIN {X 0,Y 365.975,Z 575.297,A -85,B 0,C 180,E1 11879.998,E2 11879.998} C_VEL
LIN {X 0,Y 365.994,Z 571.57,A -85,B 0,C 180,E1 11884.744,E2 11884.744} C_VEL
LIN {X 0,Y 366.656,Z 562.747,A -85,B 0,C 180,E1 11889.505,E2 11889.505} C_VEL
LIN {X 0,Y 367.956,Z 548.306,A -85,B 0,C 180,E1 11894.29,E2 11894.29} C_VEL
LIN {X 0,Y 370.372,Z 528.224,A -85,B 0,C 180,E1 11898.776,E2 11898.776} C_VEL
LIN {X 0,Y 373.516,Z 502.563,A -85,B 0,C 180,E1 11902.802,E2 11902.802} C_VEL
LIN {X 0,Y 376.881,Z 473.081,A -85,B 0,C 180,E1 11906.064,E2 11906.064} C_VEL
LIN {X 0,Y 380.059,Z 440.144,A -85,B 0,C 180,E1 11908.553,E2 11908.553} C_VEL
LIN {X 0,Y 380.605,Z 422.736,A -85,B 0,C 180,E1 11909.534,E2 11909.534} C_VEL
LIN {X 0,Y 369.02,Z 386.143,A -85,B 0,C 180,E1 11911.677,E2 11911.677} C_VEL
LIN {X 0,Y 363.644,Z 370.16,A -85,B 0,C 180,E1 11912.51,E2 11912.51} C_VEL
LIN {X 0,Y 363.432,Z 370.16,A -85,B 0,C 180,E1 11918.668,E2 11918.668} C_VEL
LIN {X 0,Y 363.381,Z 370.16,A -85,B 0,C 180,E1 11925.09,E2 11925.09} C_VEL
LIN {X 0,Y 363.405,Z 370.947,A -85,B 0,C 180,E1 11931.575,E2 11931.575} C_VEL
LIN {X 0,Y 382.161,Z 408.105,A -85,B 0,C 180,E1 11935.034,E2 11935.034} C_VEL
LIN {X 0,Y 392.625,Z 437.95,A -85,B 0,C 180,E1 11937.86,E2 11937.86} C_VEL
LIN {X 0,Y 387.922,Z 469.939,A -85,B 0,C 180,E1 11940.163,E2 11940.163} C_VEL
LIN {X 0,Y 382.551,Z 497.812,A -85,B 0,C 180,E1 11943.152,E2 11943.152} C_VEL
LIN {X 0,Y 377.024,Z 522.381,A -85,B 0,C 180,E1 11946.888,E2 11946.888} C_VEL
LIN {X 0,Y 372.221,Z 542.776,A -85,B 0,C 180,E1 11951.323,E2 11951.323} C_VEL
LIN {X 0,Y 368.676,Z 558.538,A -85,B 0,C 180,E1 11956.346,E2 11956.346} C_VEL
LIN {X 0,Y 366.732,Z 568.963,A -85,B 0,C 180,E1 11961.687,E2 11961.687} C_VEL
LIN {X 0,Y 366.175,Z 572.943,A -85,B 0,C 180,E1 11965.26,E2 11965.26} C_VEL
LIN {X 0,Y 365.824,Z 574.795,A -85,B 0,C 180,E1 11970.004,E2 11970.004} C_VEL
LIN {X 0,Y 366.317,Z 571.745,A -85,B 0,C 180,E1 11975.934,E2 11975.934} C_VEL
LIN {X 0,Y 367.668,Z 563.673,A -85,B 0,C 180,E1 11981.283,E2 11981.283} C_VEL
LIN {X 0,Y 370.559,Z 549.745,A -85,B 0,C 180,E1 11986.621,E2 11986.621} C_VEL
LIN {X 0,Y 374.937,Z 531.056,A -85,B 0,C 180,E1 11991.313,E2 11991.313} C_VEL
LIN {X 0,Y 380.515,Z 507.125,A -85,B 0,C 180,E1 11995.483,E2 11995.483} C_VEL
LIN {X 0,Y 386.226,Z 479.182,A -85,B 0,C 180,E1 11998.861,E2 11998.861} C_VEL
LIN {X 0,Y 391.256,Z 448.171,A -85,B 0,C 180,E1 12001.411,E2 12001.411} C_VEL
LIN {X 0,Y 392.244,Z 436.878,A -85,B 0,C 180,E1 12002.148,E2 12002.148} C_VEL
LIN {X 0,Y 381.158,Z 405.906,A -85,B 0,C 180,E1 12005.072,E2 12005.072} C_VEL
LIN {X 0,Y 365.001,Z 375.039,A -85,B 0,C 180,E1 12007.998,E2 12007.998} C_VEL
LIN {X 0,Y 363.31,Z 370.16,A -85,B 0,C 180,E1 12008.412,E2 12008.412} C_VEL
LIN {X 0,Y 363.343,Z 370.16,A -85,B 0,C 180,E1 12015.105,E2 12015.105} C_VEL
LIN {X 0,Y 363.36,Z 370.16,A -85,B 0,C 180,E1 12022.344,E2 12022.344} C_VEL
LIN {X 0,Y 363.583,Z 370.16,A -85,B 0,C 180,E1 12030.024,E2 12030.024} C_VEL
LIN {X 0,Y 363.865,Z 370.16,A -85,B 0,C 180,E1 12038.011,E2 12038.011} C_VEL
LIN {X 0,Y 364.284,Z 370.16,A -85,B 0,C 180,E1 12045.563,E2 12045.563} C_VEL
LIN {X 0,Y 364.631,Z 370.16,A -85,B 0,C 180,E1 12052.846,E2 12052.846} C_VEL
LIN {X 0,Y 365.018,Z 370.16,A -85,B 0,C 180,E1 12060.002,E2 12060.002} C_VEL
LIN {X 0,Y 364.662,Z 370.16,A -85,B 0,C 180,E1 12067.156,E2 12067.156} C_VEL
LIN {X 0,Y 364.194,Z 370.16,A -85,B 0,C 180,E1 12074.444,E2 12074.444} C_VEL
LIN {X 0,Y 363.853,Z 370.16,A -85,B 0,C 180,E1 12081.993,E2 12081.993} C_VEL
LIN {X 0,Y 363.602,Z 370.16,A -85,B 0,C 180,E1 12089.978,E2 12089.978} C_VEL
LIN {X 0,Y 363.415,Z 370.16,A -85,B 0,C 180,E1 12097.667,E2 12097.667} C_VEL
LIN {X 0,Y 363.385,Z 370.16,A -85,B 0,C 180,E1 12105.094,E2 12105.094} C_VEL
LIN {X 0,Y 363.433,Z 370.278,A -85,B 0,C 180,E1 12106.491,E2 12106.491} C_VEL
LIN {X 0,Y 368.1,Z 380.276,A -85,B 0,C 180,E1 12107.384,E2 12107.384} C_VEL
LIN {X 0,Y 386.609,Z 417.845,A -85,B 0,C 180,E1 12110.609,E2 12110.609} C_VEL
LIN {X 0,Y 393.848,Z 439.425,A -85,B 0,C 180,E1 12112.229,E2 12112.229} C_VEL
LIN {X 0,Y 389.391,Z 476.931,A -85,B 0,C 180,E1 12114.082,E2 12114.082} C_VEL
LIN {X 0,Y 384.161,Z 510.807,A -85,B 0,C 180,E1 12116.68,E2 12116.68} C_VEL
LIN {X 0,Y 378.453,Z 542.711,A -85,B 0,C 180,E1 12120.159,E2 12120.159} C_VEL
LIN {X 0,Y 373.101,Z 571.01,A -85,B 0,C 180,E1 12124.457,E2 12124.457} C_VEL
LIN {X 0,Y 369.146,Z 594.208,A -85,B 0,C 180,E1 12129.281,E2 12129.281} C_VEL
LIN {X 0,Y 366.793,Z 612.052,A -85,B 0,C 180,E1 12134.434,E2 12134.434} C_VEL
LIN {X 0,Y 365.771,Z 624.729,A -85,B 0,C 180,E1 12139.865,E2 12139.865} C_VEL
LIN {X 0,Y 365.522,Z 631.894,A -85,B 0,C 180,E1 12145.245,E2 12145.245} C_VEL
LIN {X 0,Y 365.54,Z 633.97,A -85,B 0,C 180,E1 12149.996,E2 12149.996} C_VEL
LIN {X 0,Y 365.506,Z 631.902,A -85,B 0,C 180,E1 12154.748,E2 12154.748} C_VEL
LIN {X 0,Y 365.771,Z 624.745,A -85,B 0,C 180,E1 12160.128,E2 12160.128} C_VEL
LIN {X 0,Y 365.868,Z 622.554,A -85,B 0,C 180,E1 12161.257,E2 12161.257} C_VEL
LIN {X 0,Y 364.815,Z 619.796,A -85,B 0,C 180,E1 12162.549,E2 12162.549} C_VEL
LIN {X 0,Y 359.187,Z 611.055,A -85,B 0,C 180,E1 12166.024,E2 12166.024} C_VEL
LIN {X 0,Y 359.206,Z 610.099,A -85,B 0,C 180,E1 12166.342,E2 12166.342} C_VEL
LIN {X 0,Y 362.031,Z 590.997,A -85,B 0,C 180,E1 12171.782,E2 12171.782} C_VEL
LIN {X 0,Y 366.47,Z 566.969,A -85,B 0,C 180,E1 12176.692,E2 12176.692} C_VEL
LIN {X 0,Y 372.177,Z 537.604,A -85,B 0,C 180,E1 12181.016,E2 12181.016} C_VEL
LIN {X 0,Y 378.124,Z 505.562,A -85,B 0,C 180,E1 12184.406,E2 12184.406} C_VEL
LIN {X 0,Y 383.806,Z 469.745,A -85,B 0,C 180,E1 12186.998,E2 12186.998} C_VEL
LIN {X 0,Y 386.904,Z 439.41,A -85,B 0,C 180,E1 12188.501,E2 12188.501} C_VEL
LIN {X 0,Y 375.013,Z 408.61,A -85,B 0,C 180,E1 12191.013,E2 12191.013} C_VEL
LIN {X 0,Y 361.583,Z 382.122,A -85,B 0,C 180,E1 12193.574,E2 12193.574} C_VEL
LIN {X 0,Y 361.222,Z 378.786,A -85,B 0,C 180,E1 12195.105,E2 12195.105} C_VEL
LIN {X 0,Y 361.231,Z 378.428,A -85,B 0,C 180,E1 12196.955,E2 12196.955} C_VEL
LIN {X 0,Y 365.269,Z 385.559,A -85,B 0,C 180,E1 12201.183,E2 12201.183} C_VEL
LIN {X 0,Y 371.282,Z 395.975,A -85,B 0,C 180,E1 12203.915,E2 12203.915} C_VEL
LIN {X 0,Y 378.424,Z 412.513,A -85,B 0,C 180,E1 12206.353,E2 12206.353} C_VEL
LIN {X 0,Y 382.326,Z 429.158,A -85,B 0,C 180,E1 12207.987,E2 12207.987} C_VEL
LIN {X 0,Y 378.104,Z 464.129,A -85,B 0,C 180,E1 12210.217,E2 12210.217} C_VEL
LIN {X 0,Y 373.376,Z 495.335,A -85,B 0,C 180,E1 12213.218,E2 12213.218} C_VEL
LIN {X 0,Y 368.428,Z 522.689,A -85,B 0,C 180,E1 12217.021,E2 12217.021} C_VEL
LIN {X 0,Y 364.444,Z 543.644,A -85,B 0,C 180,E1 12221.218,E2 12221.218} C_VEL
LIN {X 0,Y 361.132,Z 560.116,A -85,B 0,C 180,E1 12226.05,E2 12226.05} C_VEL
LIN {X 0,Y 359.233,Z 570.732,A -85,B 0,C 180,E1 12231.115,E2 12231.115} C_VEL
LIN {X 0,Y 358.512,Z 575.128,A -85,B 0,C 180,E1 12235.154,E2 12235.154} C_VEL
LIN {X 0,Y 358.129,Z 575.963,A -85,B 0,C 180,E1 12239.998,E2 12239.998} C_VEL
LIN {X 0,Y 358.123,Z 572.073,A -85,B 0,C 180,E1 12244.848,E2 12244.848} C_VEL
LIN {X 0,Y 358.823,Z 563.039,A -85,B 0,C 180,E1 12249.714,E2 12249.714} C_VEL
LIN {X 0,Y 360.221,Z 548.297,A -85,B 0,C 180,E1 12254.604,E2 12254.604} C_VEL
LIN {X 0,Y 362.766,Z 527.876,A -85,B 0,C 180,E1 12259.185,E2 12259.185} C_VEL
LIN {X 0,Y 366.089,Z 501.769,A -85,B 0,C 180,E1 12263.292,E2 12263.292} C_VEL
LIN {X 0,Y 369.679,Z 471.409,A -85,B 0,C 180,E1 12266.639,E2 12266.639} C_VEL
LIN {X 0,Y 372.929,Z 437.737,A -85,B 0,C 180,E1 12269.151,E2 12269.151} C_VEL
LIN {X 0,Y 373.117,Z 424.181,A -85,B 0,C 180,E1 12269.929,E2 12269.929} C_VEL
LIN {X 0,Y 362.106,Z 389.089,A -85,B 0,C 180,E1 12272.059,E2 12272.059} C_VEL
LIN {X 0,Y 355.678,Z 370.16,A -85,B 0,C 180,E1 12273.121,E2 12273.121} C_VEL
LIN {X 0,Y 355.43,Z 370.16,A -85,B 0,C 180,E1 12279.947,E2 12279.947} C_VEL
LIN {X 0,Y 355.38,Z 370.16,A -85,B 0,C 180,E1 12287.036,E2 12287.036} C_VEL
LIN {X 0,Y 355.458,Z 370.797,A -85,B 0,C 180,E1 12290.449,E2 12290.449} C_VEL
LIN {X 0,Y 374.815,Z 408.536,A -85,B 0,C 180,E1 12294.179,E2 12294.179} C_VEL
LIN {X 0,Y 385.33,Z 438.346,A -85,B 0,C 180,E1 12297.115,E2 12297.115} C_VEL
LIN {X 0,Y 384.801,Z 448.295,A -85,B 0,C 180,E1 12297.821,E2 12297.821} C_VEL
LIN {X 0,Y 379.533,Z 479.596,A -85,B 0,C 180,E1 12300.424,E2 12300.424} C_VEL
LIN {X 0,Y 373.569,Z 507.572,A -85,B 0,C 180,E1 12303.854,E2 12303.854} C_VEL
LIN {X 0,Y 367.938,Z 530.432,A -85,B 0,C 180,E1 12307.856,E2 12307.856} C_VEL
LIN {X 0,Y 363.395,Z 548.769,A -85,B 0,C 180,E1 12312.424,E2 12312.424} C_VEL
LIN {X 0,Y 360.104,Z 563.297,A -85,B 0,C 180,E1 12317.869,E2 12317.869} C_VEL
LIN {X 0,Y 358.666,Z 571.168,A -85,B 0,C 180,E1 12322.729,E2 12322.729} C_VEL
LIN {X 0,Y 357.959,Z 574.943,A -85,B 0,C 180,E1 12327.58,E2 12327.58} C_VEL
LIN {X 0,Y 357.975,Z 574.899,A -85,B 0,C 180,E1 12332.427,E2 12332.427} C_VEL
LIN {X 0,Y 358.697,Z 571.036,A -85,B 0,C 180,E1 12337.278,E2 12337.278} C_VEL
LIN {X 0,Y 360.409,Z 561.812,A -85,B 0,C 180,E1 12342.744,E2 12342.744} C_VEL
LIN {X 0,Y 363.75,Z 547.374,A -85,B 0,C 180,E1 12347.879,E2 12347.879} C_VEL
LIN {X 0,Y 368.58,Z 527.777,A -85,B 0,C 180,E1 12352.591,E2 12352.591} C_VEL
LIN {X 0,Y 374.483,Z 503.128,A -85,B 0,C 180,E1 12356.68,E2 12356.68} C_VEL
LIN {X 0,Y 380.54,Z 474.273,A -85,B 0,C 180,E1 12359.99,E2 12359.99} C_VEL
LIN {X 0,Y 385.559,Z 442.683,A -85,B 0,C 180,E1 12362.443,E2 12362.443} C_VEL
LIN {X 0,Y 383.138,Z 431.179,A -85,B 0,C 180,E1 12363.511,E2 12363.511} C_VEL
LIN {X 0,Y 371.511,Z 401.479,A -85,B 0,C 180,E1 12366.411,E2 12366.411} C_VEL
LIN {X 0,Y 355.471,Z 371.448,A -85,B 0,C 180,E1 12369.417,E2 12369.417} C_VEL
LIN {X 0,Y 355.352,Z 370.16,A -85,B 0,C 180,E1 12369.478,E2 12369.478} C_VEL
LIN {X 0,Y 355.349,Z 370.16,A -85,B 0,C 180,E1 12377.029,E2 12377.029} C_VEL
LIN {X 0,Y 355.443,Z 370.16,A -85,B 0,C 180,E1 12384.03,E2 12384.03} C_VEL
LIN {X 0,Y 355.717,Z 370.16,A -85,B 0,C 180,E1 12392.087,E2 12392.087} C_VEL
LIN {X 0,Y 356.069,Z 370.16,A -85,B 0,C 180,E1 12400.116,E2 12400.116} C_VEL
LIN {X 0,Y 356.457,Z 370.16,A -85,B 0,C 180,E1 12407.741,E2 12407.741} C_VEL
LIN {X 0,Y 356.9,Z 370.16,A -85,B 0,C 180,E1 12415.135,E2 12415.135} C_VEL
LIN {X 0,Y 357.071,Z 370.16,A -85,B 0,C 180,E1 12422.432,E2 12422.432} C_VEL
LIN {X 0,Y 356.495,Z 370.16,A -85,B 0,C 180,E1 12429.782,E2 12429.782} C_VEL
LIN {X 0,Y 356.185,Z 370.16,A -85,B 0,C 180,E1 12437.311,E2 12437.311} C_VEL
LIN {X 0,Y 355.758,Z 370.16,A -85,B 0,C 180,E1 12445.187,E2 12445.187} C_VEL
LIN {X 0,Y 355.519,Z 370.16,A -85,B 0,C 180,E1 12451.599,E2 12451.599} C_VEL
LIN {X 0,Y 355.471,Z 370.16,A -85,B 0,C 180,E1 12456.603,E2 12456.603} C_VEL
LIN {X 0,Y 355.374,Z 370.16,A -85,B 0,C 180,E1 12463.591,E2 12463.591} C_VEL
LIN {X 0,Y 355.536,Z 370.715,A -85,B 0,C 180,E1 12465.395,E2 12465.395} C_VEL
LIN {X 0,Y 378.312,Z 416.094,A -85,B 0,C 180,E1 12469.617,E2 12469.617} C_VEL
LIN {X 0,Y 387.112,Z 440.533,A -85,B 0,C 180,E1 12471.584,E2 12471.584} C_VEL
LIN {X 0,Y 382.635,Z 477.579,A -85,B 0,C 180,E1 12473.489,E2 12473.489} C_VEL
LIN {X 0,Y 377.119,Z 511.437,A -85,B 0,C 180,E1 12476.147,E2 12476.147} C_VEL
LIN {X 0,Y 370.995,Z 543.787,A -85,B 0,C 180,E1 12479.79,E2 12479.79} C_VEL
LIN {X 0,Y 365.43,Z 571.926,A -85,B 0,C 180,E1 12484.211,E2 12484.211} C_VEL
LIN {X 0,Y 361.121,Z 595.914,A -85,B 0,C 180,E1 12489.441,E2 12489.441} C_VEL
LIN {X 0,Y 358.787,Z 613.015,A -85,B 0,C 180,E1 12494.705,E2 12494.705} C_VEL
LIN {X 0,Y 357.842,Z 625.114,A -85,B 0,C 180,E1 12500.253,E2 12500.253} C_VEL
LIN {X 0,Y 357.661,Z 631.253,A -85,B 0,C 180,E1 12505.14,E2 12505.14} C_VEL
LIN {X 0,Y 357.684,Z 633.334,A -85,B 0,C 180,E1 12509.996,E2 12509.996} C_VEL
LIN {X 0,Y 357.645,Z 631.262,A -85,B 0,C 180,E1 12514.853,E2 12514.853} C_VEL
LIN {X 0,Y 357.918,Z 624.087,A -85,B 0,C 180,E1 12520.353,E2 12520.353} C_VEL
LIN {X 0,Y 359.062,Z 611.403,A -85,B 0,C 180,E1 12525.902,E2 12525.902} C_VEL
LIN {X 0,Y 359.206,Z 610.099,A -85,B 0,C 180,E1 12526.342,E2 12526.342} C_VEL
LIN {X 0,Y 356.289,Z 602.566,A -85,B 0,C 180,E1 12528.83,E2 12528.83} C_VEL
LIN {X 0,Y 353.747,Z 594.212,A -85,B 0,C 180,E1 12531.295,E2 12531.295} C_VEL
LIN {X 0,Y 358.128,Z 571.255,A -85,B 0,C 180,E1 12536.347,E2 12536.347} C_VEL
LIN {X 0,Y 363.784,Z 543.544,A -85,B 0,C 180,E1 12540.792,E2 12540.792} C_VEL
LIN {X 0,Y 370.293,Z 510.666,A -85,B 0,C 180,E1 12544.556,E2 12544.556} C_VEL
LIN {X 0,Y 376.222,Z 476.719,A -85,B 0,C 180,E1 12547.231,E2 12547.231} C_VEL
LIN {X 0,Y 380.193,Z 441.294,A -85,B 0,C 180,E1 12549.132,E2 12549.132} C_VEL
LIN {X 0,Y 368.189,Z 410.229,A -85,B 0,C 180,E1 12551.807,E2 12551.807} C_VEL
LIN {X 0,Y 358.968,Z 391.297,A -85,B 0,C 180,E1 12553.716,E2 12553.716} C_VEL
LIN {X 0,Y 359.191,Z 387.023,A -85,B 0,C 180,E1 12554.792,E2 12554.792} C_VEL
LIN {X 0,Y 359.138,Z 386.165,A -85,B 0,C 180,E1 12556.882,E2 12556.882} C_VEL
LIN {X 0,Y 362.567,Z 393.057,A -85,B 0,C 180,E1 12560.916,E2 12560.916} C_VEL
LIN {X 0,Y 367.914,Z 402.988,A -85,B 0,C 180,E1 12563.556,E2 12563.556} C_VEL
LIN {X 0,Y 374.259,Z 419.604,A -85,B 0,C 180,E1 12566.021,E2 12566.021} C_VEL
LIN {X 0,Y 376.352,Z 433.302,A -85,B 0,C 180,E1 12567.335,E2 12567.335} C_VEL
LIN {X 0,Y 371.593,Z 468.302,A -85,B 0,C 180,E1 12569.722,E2 12569.722} C_VEL
LIN {X 0,Y 366.219,Z 499.792,A -85,B 0,C 180,E1 12572.951,E2 12572.951} C_VEL
LIN {X 0,Y 360.952,Z 526.249,A -85,B 0,C 180,E1 12576.878,E2 12576.878} C_VEL
LIN {X 0,Y 356.85,Z 546.277,A -85,B 0,C 180,E1 12581.125,E2 12581.125} C_VEL
LIN {X 0,Y 353.527,Z 561.291,A -85,B 0,C 180,E1 12585.744,E2 12585.744} C_VEL
LIN {X 0,Y 351.761,Z 570.44,A -85,B 0,C 180,E1 12590.085,E2 12590.085} C_VEL
LIN {X 0,Y 350.697,Z 575.959,A -85,B 0,C 180,E1 12595.045,E2 12595.045} C_VEL
LIN {X 0,Y 350.28,Z 576.634,A -85,B 0,C 180,E1 12599.998,E2 12599.998} C_VEL
LIN {X 0,Y 350.252,Z 572.53,A -85,B 0,C 180,E1 12604.958,E2 12604.958} C_VEL
LIN {X 0,Y 350.987,Z 563.278,A -85,B 0,C 180,E1 12609.933,E2 12609.933} C_VEL
LIN {X 0,Y 352.484,Z 548.232,A -85,B 0,C 180,E1 12614.932,E2 12614.932} C_VEL
LIN {X 0,Y 355.171,Z 527.428,A -85,B 0,C 180,E1 12619.612,E2 12619.612} C_VEL
LIN {X 0,Y 358.517,Z 502.011,A -85,B 0,C 180,E1 12623.649,E2 12623.649} C_VEL
LIN {X 0,Y 362.222,Z 471.715,A -85,B 0,C 180,E1 12627.039,E2 12627.039} C_VEL
LIN {X 0,Y 365.602,Z 437.953,A -85,B 0,C 180,E1 12629.596,E2 12629.596} C_VEL
LIN {X 0,Y 365.625,Z 425.469,A -85,B 0,C 180,E1 12630.339,E2 12630.339} C_VEL
LIN {X 0,Y 354.136,Z 388.944,A -85,B 0,C 180,E1 12632.62,E2 12632.62} C_VEL
LIN {X 0,Y 347.739,Z 370.16,A -85,B 0,C 180,E1 12633.721,E2 12633.721} C_VEL
LIN {X 0,Y 347.42,Z 370.16,A -85,B 0,C 180,E1 12640.814,E2 12640.814} C_VEL
LIN {X 0,Y 347.393,Z 370.16,A -85,B 0,C 180,E1 12647.801,E2 12647.801} C_VEL
LIN {X 0,Y 347.422,Z 370.555,A -85,B 0,C 180,E1 12649.235,E2 12649.235} C_VEL
LIN {X 0,Y 350.229,Z 376.126,A -85,B 0,C 180,E1 12649.807,E2 12649.807} C_VEL
LIN {X 0,Y 367.55,Z 409.402,A -85,B 0,C 180,E1 12653.309,E2 12653.309} C_VEL
LIN {X 0,Y 378.199,Z 439.253,A -85,B 0,C 180,E1 12656.39,E2 12656.39} C_VEL
LIN {X 0,Y 378.626,Z 446.689,A -85,B 0,C 180,E1 12657.018,E2 12657.018} C_VEL
LIN {X 0,Y 373.31,Z 477.676,A -85,B 0,C 180,E1 12659.545,E2 12659.545} C_VEL
LIN {X 0,Y 367.36,Z 504.737,A -85,B 0,C 180,E1 12662.794,E2 12662.794} C_VEL
LIN {X 0,Y 361.123,Z 529.291,A -85,B 0,C 180,E1 12666.988,E2 12666.988} C_VEL
LIN {X 0,Y 356.141,Z 548.406,A -85,B 0,C 180,E1 12671.733,E2 12671.733} C_VEL
LIN {X 0,Y 352.659,Z 562.696,A -85,B 0,C 180,E1 12676.979,E2 12676.979} C_VEL
LIN {X 0,Y 350.836,Z 571.809,A -85,B 0,C 180,E1 12682.566,E2 12682.566} C_VEL
LIN {X 0,Y 350.089,Z 575.581,A -85,B 0,C 180,E1 12687.525,E2 12687.525} C_VEL
LIN {X 0,Y 350.105,Z 575.537,A -85,B 0,C 180,E1 12692.482,E2 12692.482} C_VEL
LIN {X 0,Y 350.89,Z 571.677,A -85,B 0,C 180,E1 12697.441,E2 12697.441} C_VEL
LIN {X 0,Y 352.705,Z 562.465,A -85,B 0,C 180,E1 12703.027,E2 12703.027} C_VEL
LIN {X 0,Y 356.224,Z 548.045,A -85,B 0,C 180,E1 12708.27,E2 12708.27} C_VEL
LIN {X 0,Y 361.362,Z 528.196,A -85,B 0,C 180,E1 12713.13,E2 12713.13} C_VEL
LIN {X 0,Y 367.476,Z 503.882,A -85,B 0,C 180,E1 12717.231,E2 12717.231} C_VEL
LIN {X 0,Y 373.759,Z 475.15,A -85,B 0,C 180,E1 12720.591,E2 12720.591} C_VEL
LIN {X 0,Y 379.009,Z 443.553,A -85,B 0,C 180,E1 12723.089,E2 12723.089} C_VEL
LIN {X 0,Y 370.114,Z 415.549,A -85,B 0,C 180,E1 12725.962,E2 12725.962} C_VEL
LIN {X 0,Y 355.339,Z 385.558,A -85,B 0,C 180,E1 12729.089,E2 12729.089} C_VEL
LIN {X 0,Y 347.443,Z 371.257,A -85,B 0,C 180,E1 12730.626,E2 12730.626} C_VEL
LIN {X 0,Y 347.333,Z 370.16,A -85,B 0,C 180,E1 12730.834,E2 12730.834} C_VEL
LIN {X 0,Y 347.362,Z 370.16,A -85,B 0,C 180,E1 12737.816,E2 12737.816} C_VEL
LIN {X 0,Y 347.522,Z 370.16,A -85,B 0,C 180,E1 12745.871,E2 12745.871} C_VEL
LIN {X 0,Y 347.695,Z 370.16,A -85,B 0,C 180,E1 12751.385,E2 12751.385} C_VEL
LIN {X 0,Y 348.118,Z 370.16,A -85,B 0,C 180,E1 12759.642,E2 12759.642} C_VEL
LIN {X 0,Y 348.379,Z 370.16,A -85,B 0,C 180,E1 12764.888,E2 12764.888} C_VEL
LIN {X 0,Y 348.769,Z 370.16,A -85,B 0,C 180,E1 12772.519,E2 12772.519} C_VEL
LIN {X 0,Y 349.227,Z 370.16,A -85,B 0,C 180,E1 12780.002,E2 12780.002} C_VEL
LIN {X 0,Y 348.787,Z 370.16,A -85,B 0,C 180,E1 12787.484,E2 12787.484} C_VEL
LIN {X 0,Y 348.293,Z 370.16,A -85,B 0,C 180,E1 12795.119,E2 12795.119} C_VEL
LIN {X 0,Y 348.1,Z 370.16,A -85,B 0,C 180,E1 12800.362,E2 12800.362} C_VEL
LIN {X 0,Y 347.707,Z 370.16,A -85,B 0,C 180,E1 12808.618,E2 12808.618} C_VEL
LIN {X 0,Y 347.57,Z 370.16,A -85,B 0,C 180,E1 12814.49,E2 12814.49} C_VEL
LIN {X 0,Y 347.4,Z 370.16,A -85,B 0,C 180,E1 12822.191,E2 12822.191} C_VEL
LIN {X 0,Y 347.516,Z 370.51,A -85,B 0,C 180,E1 12824.191,E2 12824.191} C_VEL
LIN {X 0,Y 352.781,Z 380.861,A -85,B 0,C 180,E1 12825.285,E2 12825.285} C_VEL
LIN {X 0,Y 371.039,Z 416.64,A -85,B 0,C 180,E1 12828.762,E2 12828.762} C_VEL
LIN {X 0,Y 380.475,Z 443.74,A -85,B 0,C 180,E1 12831.045,E2 12831.045} C_VEL
LIN {X 0,Y 375.735,Z 479.368,A -85,B 0,C 180,E1 12832.949,E2 12832.949} C_VEL
LIN {X 0,Y 369.834,Z 513.628,A -85,B 0,C 180,E1 12835.742,E2 12835.742} C_VEL
LIN {X 0,Y 363.494,Z 545.268,A -85,B 0,C 180,E1 12839.463,E2 12839.463} C_VEL
LIN {X 0,Y 357.767,Z 572.846,A -85,B 0,C 180,E1 12843.954,E2 12843.954} C_VEL
LIN {X 0,Y 353.283,Z 596.357,A -85,B 0,C 180,E1 12849.292,E2 12849.292} C_VEL
LIN {X 0,Y 350.799,Z 613.979,A -85,B 0,C 180,E1 12854.989,E2 12854.989} C_VEL
LIN {X 0,Y 349.969,Z 624.455,A -85,B 0,C 180,E1 12860.032,E2 12860.032} C_VEL
LIN {X 0,Y 349.776,Z 630.609,A -85,B 0,C 180,E1 12865.03,E2 12865.03} C_VEL
LIN {X 0,Y 349.807,Z 632.697,A -85,B 0,C 180,E1 12869.996,E2 12869.996} C_VEL
LIN {X 0,Y 349.758,Z 630.289,A -85,B 0,C 180,E1 12875.396,E2 12875.396} C_VEL
LIN {X 0,Y 350.09,Z 622.312,A -85,B 0,C 180,E1 12881.217,E2 12881.217} C_VEL
LIN {X 0,Y 351.484,Z 608.876,A -85,B 0,C 180,E1 12886.898,E2 12886.898} C_VEL
LIN {X 0,Y 353.747,Z 594.212,A -85,B 0,C 180,E1 12891.295,E2 12891.295} C_VEL
LIN {X 0,Y 351.534,Z 585.104,A -85,B 0,C 180,E1 12893.704,E2 12893.704} C_VEL
LIN {X 0,Y 349.815,Z 575.09,A -85,B 0,C 180,E1 12896.04,E2 12896.04} C_VEL
LIN {X 0,Y 355.687,Z 548.035,A -85,B 0,C 180,E1 12900.71,E2 12900.71} C_VEL
LIN {X 0,Y 362.266,Z 517.213,A -85,B 0,C 180,E1 12904.522,E2 12904.522} C_VEL
LIN {X 0,Y 368.442,Z 484.136,A -85,B 0,C 180,E1 12907.412,E2 12907.412} C_VEL
LIN {X 0,Y 373.585,Z 448.369,A -85,B 0,C 180,E1 12909.478,E2 12909.478} C_VEL
LIN {X 0,Y 372.835,Z 440.313,A -85,B 0,C 180,E1 12910.017,E2 12910.017} C_VEL
LIN {X 0,Y 359.564,Z 408.111,A -85,B 0,C 180,E1 12913.003,E2 12913.003} C_VEL
LIN {X 0,Y 356.325,Z 400.604,A -85,B 0,C 180,E1 12913.858,E2 12913.858} C_VEL
LIN {X 0,Y 357.028,Z 394.267,A -85,B 0,C 180,E1 12915.217,E2 12915.217} C_VEL
LIN {X 0,Y 357.015,Z 394.16,A -85,B 0,C 180,E1 12916.999,E2 12916.999} C_VEL
LIN {X 0,Y 359.922,Z 400.491,A -85,B 0,C 180,E1 12920.636,E2 12920.636} C_VEL
LIN {X 0,Y 364.543,Z 409.819,A -85,B 0,C 180,E1 12923.15,E2 12923.15} C_VEL
LIN {X 0,Y 369.808,Z 426.077,A -85,B 0,C 180,E1 12925.614,E2 12925.614} C_VEL
LIN {X 0,Y 370.786,Z 435.411,A -85,B 0,C 180,E1 12926.527,E2 12926.527} C_VEL
LIN {X 0,Y 365.473,Z 470.287,A -85,B 0,C 180,E1 12929.005,E2 12929.005} C_VEL
LIN {X 0,Y 359.744,Z 501.134,A -85,B 0,C 180,E1 12932.27,E2 12932.27} C_VEL
LIN {X 0,Y 354.333,Z 526.265,A -85,B 0,C 180,E1 12936.051,E2 12936.051} C_VEL
LIN {X 0,Y 349.514,Z 547.756,A -85,B 0,C 180,E1 12940.713,E2 12940.713} C_VEL
LIN {X 0,Y 345.945,Z 562.539,A -85,B 0,C 180,E1 12945.424,E2 12945.424} C_VEL
LIN {X 0,Y 344.042,Z 571.5,A -85,B 0,C 180,E1 12949.861,E2 12949.861} C_VEL
LIN {X 0,Y 342.873,Z 576.796,A -85,B 0,C 180,E1 12954.932,E2 12954.932} C_VEL
LIN {X 0,Y 342.426,Z 577.303,A -85,B 0,C 180,E1 12959.998,E2 12959.998} C_VEL
LIN {X 0,Y 342.41,Z 572.974,A -85,B 0,C 180,E1 12965.071,E2 12965.071} C_VEL
LIN {X 0,Y 343.143,Z 563.503,A -85,B 0,C 180,E1 12970.163,E2 12970.163} C_VEL
LIN {X 0,Y 344.775,Z 548.121,A -85,B 0,C 180,E1 12975.274,E2 12975.274} C_VEL
LIN {X 0,Y 347.607,Z 526.898,A -85,B 0,C 180,E1 12980.056,E2 12980.056} C_VEL
LIN {X 0,Y 351.098,Z 500.93,A -85,B 0,C 180,E1 12984.18,E2 12984.18} C_VEL
LIN {X 0,Y 354.934,Z 470.262,A -85,B 0,C 180,E1 12987.6,E2 12987.6} C_VEL
LIN {X 0,Y 358.359,Z 436.593,A -85,B 0,C 180,E1 12990.136,E2 12990.136} C_VEL
LIN {X 0,Y 358.174,Z 426.907,A -85,B 0,C 180,E1 12990.74,E2 12990.74} C_VEL
LIN {X 0,Y 346.768,Z 390.472,A -85,B 0,C 180,E1 12993.11,E2 12993.11} C_VEL
LIN {X 0,Y 339.762,Z 370.16,A -85,B 0,C 180,E1 12994.323,E2 12994.323} C_VEL
LIN {X 0,Y 339.494,Z 370.16,A -85,B 0,C 180,E1 13001.98,E2 13001.98} C_VEL
LIN {X 0,Y 339.5,Z 370.16,A -85,B 0,C 180,E1 13007.909,E2 13007.909} C_VEL
LIN {X 0,Y 342.101,Z 376.029,A -85,B 0,C 180,E1 13008.534,E2 13008.534} C_VEL
LIN {X 0,Y 359.665,Z 408.706,A -85,B 0,C 180,E1 13012.234,E2 13012.234} C_VEL
LIN {X 0,Y 370.51,Z 437.957,A -85,B 0,C 180,E1 13015.398,E2 13015.398} C_VEL
LIN {X 0,Y 372.236,Z 446.739,A -85,B 0,C 180,E1 13016.296,E2 13016.296} C_VEL
LIN {X 0,Y 366.84,Z 477.041,A -85,B 0,C 180,E1 13018.776,E2 13018.776} C_VEL
LIN {X 0,Y 360.392,Z 505.33,A -85,B 0,C 180,E1 13022.197,E2 13022.197} C_VEL
LIN {X 0,Y 354.02,Z 529.418,A -85,B 0,C 180,E1 13026.369,E2 13026.369} C_VEL
LIN {X 0,Y 348.642,Z 549.072,A -85,B 0,C 180,E1 13031.326,E2 13031.326} C_VEL
LIN {X 0,Y 344.963,Z 563.343,A -85,B 0,C 180,E1 13036.683,E2 13036.683} C_VEL
LIN {X 0,Y 343.015,Z 572.449,A -85,B 0,C 180,E1 13042.395,E2 13042.395} C_VEL
LIN {X 0,Y 342.219,Z 576.218,A -85,B 0,C 180,E1 13047.468,E2 13047.468} C_VEL
LIN {X 0,Y 342.236,Z 576.174,A -85,B 0,C 180,E1 13052.539,E2 13052.539} C_VEL
LIN {X 0,Y 343.073,Z 572.318,A -85,B 0,C 180,E1 13057.611,E2 13057.611} C_VEL
LIN {X 0,Y 345.008,Z 563.118,A -85,B 0,C 180,E1 13063.323,E2 13063.323} C_VEL
LIN {X 0,Y 349.027,Z 547.684,A -85,B 0,C 180,E1 13068.989,E2 13068.989} C_VEL
LIN {X 0,Y 354.511,Z 527.364,A -85,B 0,C 180,E1 13073.939,E2 13073.939} C_VEL
LIN {X 0,Y 361.086,Z 502.278,A -85,B 0,C 180,E1 13078.146,E2 13078.146} C_VEL
LIN {X 0,Y 367.297,Z 474.521,A -85,B 0,C 180,E1 13081.362,E2 13081.362} C_VEL
LIN {X 0,Y 372.232,Z 444.49,A -85,B 0,C 180,E1 13083.785,E2 13083.785} C_VEL
LIN {X 0,Y 361.984,Z 414.01,A -85,B 0,C 180,E1 13087.085,E2 13087.085} C_VEL
LIN {X 0,Y 346.132,Z 382.954,A -85,B 0,C 180,E1 13090.527,E2 13090.527} C_VEL
LIN {X 0,Y 339.449,Z 370.85,A -85,B 0,C 180,E1 13091.919,E2 13091.919} C_VEL
LIN {X 0,Y 339.455,Z 370.16,A -85,B 0,C 180,E1 13099.31,E2 13099.31} C_VEL
LIN {X 0,Y 339.616,Z 370.16,A -85,B 0,C 180,E1 13107.663,E2 13107.663} C_VEL
LIN {X 0,Y 339.819,Z 370.16,A -85,B 0,C 180,E1 13113.546,E2 13113.546} C_VEL
LIN {X 0,Y 340.316,Z 370.16,A -85,B 0,C 180,E1 13121.858,E2 13121.858} C_VEL
LIN {X 0,Y 340.667,Z 370.16,A -85,B 0,C 180,E1 13129.763,E2 13129.763} C_VEL
LIN {X 0,Y 341.174,Z 370.16,A -85,B 0,C 180,E1 13137.458,E2 13137.458} C_VEL
LIN {X 0,Y 341.247,Z 370.16,A -85,B 0,C 180,E1 13142.544,E2 13142.544} C_VEL
LIN {X 0,Y 340.613,Z 370.16,A -85,B 0,C 180,E1 13150.243,E2 13150.243} C_VEL
LIN {X 0,Y 340.251,Z 370.16,A -85,B 0,C 180,E1 13158.149,E2 13158.149} C_VEL
LIN {X 0,Y 339.818,Z 370.16,A -85,B 0,C 180,E1 13166.457,E2 13166.457} C_VEL
LIN {X 0,Y 339.649,Z 370.16,A -85,B 0,C 180,E1 13172.337,E2 13172.337} C_VEL
LIN {X 0,Y 339.485,Z 370.16,A -85,B 0,C 180,E1 13178.634,E2 13178.634} C_VEL
LIN {X 0,Y 339.579,Z 370.16,A -85,B 0,C 180,E1 13182.86,E2 13182.86} C_VEL
LIN {X 0,Y 342.386,Z 376.183,A -85,B 0,C 180,E1 13183.554,E2 13183.554} C_VEL
LIN {X 0,Y 362.737,Z 414.735,A -85,B 0,C 180,E1 13187.65,E2 13187.65} C_VEL
LIN {X 0,Y 373.842,Z 444.695,A -85,B 0,C 180,E1 13190.36,E2 13190.36} C_VEL
LIN {X 0,Y 368.916,Z 480.942,A -85,B 0,C 180,E1 13192.374,E2 13192.374} C_VEL
LIN {X 0,Y 362.533,Z 515.605,A -85,B 0,C 180,E1 13195.317,E2 13195.317} C_VEL
LIN {X 0,Y 356.035,Z 546.534,A -85,B 0,C 180,E1 13199.09,E2 13199.09} C_VEL
LIN {X 0,Y 350.112,Z 573.726,A -85,B 0,C 180,E1 13203.686,E2 13203.686} C_VEL
LIN {X 0,Y 345.476,Z 596.805,A -85,B 0,C 180,E1 13209.138,E2 13209.138} C_VEL
LIN {X 0,Y 343.017,Z 613.301,A -85,B 0,C 180,E1 13214.64,E2 13214.64} C_VEL
LIN {X 0,Y 342.096,Z 623.797,A -85,B 0,C 180,E1 13219.8,E2 13219.8} C_VEL
LIN {X 0,Y 341.891,Z 629.967,A -85,B 0,C 180,E1 13224.915,E2 13224.915} C_VEL
LIN {X 0,Y 341.93,Z 632.06,A -85,B 0,C 180,E1 13229.996,E2 13229.996} C_VEL
LIN {X 0,Y 341.887,Z 629.978,A -85,B 0,C 180,E1 13235.077,E2 13235.077} C_VEL
LIN {X 0,Y 342.16,Z 622.77,A -85,B 0,C 180,E1 13240.835,E2 13240.835} C_VEL
LIN {X 0,Y 343.496,Z 610.037,A -85,B 0,C 180,E1 13246.644,E2 13246.644} C_VEL
LIN {X 0,Y 346.712,Z 590.844,A -85,B 0,C 180,E1 13252.458,E2 13252.458} C_VEL
LIN {X 0,Y 349.815,Z 575.09,A -85,B 0,C 180,E1 13256.04,E2 13256.04} C_VEL
LIN {X 0,Y 348.537,Z 564.457,A -85,B 0,C 180,E1 13258.32,E2 13258.32} C_VEL
LIN {X 0,Y 347.395,Z 552.992,A -85,B 0,C 180,E1 13260.504,E2 13260.504} C_VEL
LIN {X 0,Y 354.445,Z 522.053,A -85,B 0,C 180,E1 13264.649,E2 13264.649} C_VEL
LIN {X 0,Y 360.934,Z 489.156,A -85,B 0,C 180,E1 13267.734,E2 13267.734} C_VEL
LIN {X 0,Y 366.624,Z 452.964,A -85,B 0,C 180,E1 13270,E2 13270} C_VEL
LIN {X 0,Y 366.889,Z 444.808,A -85,B 0,C 180,E1 13270.46,E2 13270.46} C_VEL
LIN {X 0,Y 354.919,Z 413.987,A -85,B 0,C 180,E1 13273.45,E2 13273.45} C_VEL
LIN {X 0,Y 353.689,Z 409.679,A -85,B 0,C 180,E1 13274.053,E2 13274.053} C_VEL
LIN {X 0,Y 354.992,Z 401.161,A -85,B 0,C 180,E1 13275.886,E2 13275.886} C_VEL
LIN {X 0,Y 356.897,Z 406.482,A -85,B 0,C 180,E1 13279.933,E2 13279.933} C_VEL
LIN {X 0,Y 361.043,Z 416.181,A -85,B 0,C 180,E1 13282.653,E2 13282.653} C_VEL
LIN {X 0,Y 364.968,Z 430.695,A -85,B 0,C 180,E1 13284.953,E2 13284.953} C_VEL
LIN {X 0,Y 365.463,Z 437.837,A -85,B 0,C 180,E1 13285.688,E2 13285.688} C_VEL
LIN {X 0,Y 359.573,Z 472.363,A -85,B 0,C 180,E1 13288.243,E2 13288.243} C_VEL
LIN {X 0,Y 353.326,Z 503.012,A -85,B 0,C 180,E1 13291.6,E2 13291.6} C_VEL
LIN {X 0,Y 346.982,Z 529.922,A -85,B 0,C 180,E1 13295.854,E2 13295.854} C_VEL
LIN {X 0,Y 341.902,Z 550.43,A -85,B 0,C 180,E1 13300.602,E2 13300.602} C_VEL
LIN {X 0,Y 338.001,Z 565.289,A -85,B 0,C 180,E1 13305.737,E2 13305.737} C_VEL
LIN {X 0,Y 335.854,Z 574.308,A -85,B 0,C 180,E1 13310.921,E2 13310.921} C_VEL
LIN {X 0,Y 335.059,Z 577.651,A -85,B 0,C 180,E1 13314.814,E2 13314.814} C_VEL
LIN {X 0,Y 334.575,Z 577.971,A -85,B 0,C 180,E1 13319.998,E2 13319.998} C_VEL
LIN {X 0,Y 334.563,Z 572.997,A -85,B 0,C 180,E1 13325.465,E2 13325.465} C_VEL
LIN {X 0,Y 335.31,Z 563.708,A -85,B 0,C 180,E1 13330.403,E2 13330.403} C_VEL
LIN {X 0,Y 337.057,Z 548.015,A -85,B 0,C 180,E1 13335.632,E2 13335.632} C_VEL
LIN {X 0,Y 340.031,Z 526.368,A -85,B 0,C 180,E1 13340.523,E2 13340.523} C_VEL
LIN {X 0,Y 343.711,Z 499.85,A -85,B 0,C 180,E1 13344.734,E2 13344.734} C_VEL
LIN {X 0,Y 347.576,Z 469.779,A -85,B 0,C 180,E1 13348.094,E2 13348.094} C_VEL
LIN {X 0,Y 351.143,Z 435.585,A -85,B 0,C 180,E1 13350.675,E2 13350.675} C_VEL
LIN {X 0,Y 350.045,Z 426.085,A -85,B 0,C 180,E1 13351.336,E2 13351.336} C_VEL
LIN {X 0,Y 338.765,Z 390.339,A -85,B 0,C 180,E1 13353.695,E2 13353.695} C_VEL
LIN {X 0,Y 331.791,Z 370.16,A -85,B 0,C 180,E1 13354.915,E2 13354.915} C_VEL
LIN {X 0,Y 331.542,Z 370.16,A -85,B 0,C 180,E1 13363.228,E2 13363.228} C_VEL
LIN {X 0,Y 331.57,Z 370.611,A -85,B 0,C 180,E1 13366.597,E2 13366.597} C_VEL
LIN {X 0,Y 334.381,Z 376.198,A -85,B 0,C 180,E1 13367.247,E2 13367.247} C_VEL
LIN {X 0,Y 352.252,Z 409.01,A -85,B 0,C 180,E1 13371.21,E2 13371.21} C_VEL
LIN {X 0,Y 362.919,Z 437.143,A -85,B 0,C 180,E1 13374.401,E2 13374.401} C_VEL
LIN {X 0,Y 365.612,Z 448.675,A -85,B 0,C 180,E1 13375.678,E2 13375.678} C_VEL
LIN {X 0,Y 359.859,Z 479.345,A -85,B 0,C 180,E1 13378.277,E2 13378.277} C_VEL
LIN {X 0,Y 353.431,Z 506.074,A -85,B 0,C 180,E1 13381.601,E2 13381.601} C_VEL
LIN {X 0,Y 346.805,Z 530.111,A -85,B 0,C 180,E1 13385.846,E2 13385.846} C_VEL
LIN {X 0,Y 341.151,Z 549.737,A -85,B 0,C 180,E1 13390.9,E2 13390.9} C_VEL
LIN {X 0,Y 337.283,Z 563.989,A -85,B 0,C 180,E1 13396.374,E2 13396.374} C_VEL
LIN {X 0,Y 335.201,Z 573.09,A -85,B 0,C 180,E1 13402.217,E2 13402.217} C_VEL
LIN {X 0,Y 334.349,Z 576.855,A -85,B 0,C 180,E1 13407.409,E2 13407.409} C_VEL
LIN {X 0,Y 334.368,Z 576.812,A -85,B 0,C 180,E1 13412.599,E2 13412.599} C_VEL
LIN {X 0,Y 335.249,Z 572.96,A -85,B 0,C 180,E1 13417.79,E2 13417.79} C_VEL
LIN {X 0,Y 337.326,Z 563.769,A -85,B 0,C 180,E1 13423.632,E2 13423.632} C_VEL
LIN {X 0,Y 341.543,Z 548.352,A -85,B 0,C 180,E1 13429.421,E2 13429.421} C_VEL
LIN {X 0,Y 347.296,Z 528.069,A -85,B 0,C 180,E1 13434.468,E2 13434.468} C_VEL
LIN {X 0,Y 354.184,Z 503.032,A -85,B 0,C 180,E1 13438.745,E2 13438.745} C_VEL
LIN {X 0,Y 360.931,Z 473.885,A -85,B 0,C 180,E1 13442.157,E2 13442.157} C_VEL
LIN {X 0,Y 365.323,Z 446.02,A -85,B 0,C 180,E1 13444.477,E2 13444.477} C_VEL
LIN {X 0,Y 355.283,Z 415.953,A -85,B 0,C 180,E1 13447.894,E2 13447.894} C_VEL
LIN {X 0,Y 340.305,Z 386.487,A -85,B 0,C 180,E1 13451.357,E2 13451.357} C_VEL
LIN {X 0,Y 331.563,Z 371.253,A -85,B 0,C 180,E1 13453.263,E2 13453.263} C_VEL
LIN {X 0,Y 331.461,Z 370.16,A -85,B 0,C 180,E1 13453.338,E2 13453.338} C_VEL
LIN {X 0,Y 331.527,Z 370.16,A -85,B 0,C 180,E1 13460.93,E2 13460.93} C_VEL
LIN {X 0,Y 331.568,Z 370.16,A -85,B 0,C 180,E1 13466.778,E2 13466.778} C_VEL
LIN {X 0,Y 331.875,Z 370.16,A -85,B 0,C 180,E1 13472.862,E2 13472.862} C_VEL
LIN {X 0,Y 332.332,Z 370.16,A -85,B 0,C 180,E1 13481.407,E2 13481.407} C_VEL
LIN {X 0,Y 332.737,Z 370.16,A -85,B 0,C 180,E1 13489.516,E2 13489.516} C_VEL
LIN {X 0,Y 333.273,Z 370.16,A -85,B 0,C 180,E1 13497.398,E2 13497.398} C_VEL
LIN {X 0,Y 333.343,Z 370.16,A -85,B 0,C 180,E1 13502.605,E2 13502.605} C_VEL
LIN {X 0,Y 332.675,Z 370.16,A -85,B 0,C 180,E1 13510.49,E2 13510.49} C_VEL
LIN {X 0,Y 332.278,Z 370.16,A -85,B 0,C 180,E1 13518.6,E2 13518.6} C_VEL
LIN {X 0,Y 331.879,Z 370.16,A -85,B 0,C 180,E1 13527.142,E2 13527.142} C_VEL
LIN {X 0,Y 331.581,Z 370.16,A -85,B 0,C 180,E1 13534.724,E2 13534.724} C_VEL
LIN {X 0,Y 331.58,Z 370.278,A -85,B 0,C 180,E1 13541.545,E2 13541.545} C_VEL
LIN {X 0,Y 334.07,Z 375.899,A -85,B 0,C 180,E1 13542.162,E2 13542.162} C_VEL
LIN {X 0,Y 352.915,Z 409.774,A -85,B 0,C 180,E1 13546.151,E2 13546.151} C_VEL
LIN {X 0,Y 365.978,Z 442.248,A -85,B 0,C 180,E1 13549.298,E2 13549.298} C_VEL
LIN {X 0,Y 367.138,Z 448.746,A -85,B 0,C 180,E1 13549.812,E2 13549.812} C_VEL
LIN {X 0,Y 361.509,Z 485.687,A -85,B 0,C 180,E1 13552.013,E2 13552.013} C_VEL
LIN {X 0,Y 354.974,Z 519.014,A -85,B 0,C 180,E1 13555.029,E2 13555.029} C_VEL
LIN {X 0,Y 348.058,Z 550.262,A -85,B 0,C 180,E1 13559.078,E2 13559.078} C_VEL
LIN {X 0,Y 341.836,Z 577.094,A -85,B 0,C 180,E1 13563.947,E2 13563.947} C_VEL
LIN {X 0,Y 337.309,Z 598.986,A -85,B 0,C 180,E1 13569.475,E2 13569.475} C_VEL
LIN {X 0,Y 334.949,Z 614.82,A -85,B 0,C 180,E1 13575.208,E2 13575.208} C_VEL
LIN {X 0,Y 334.134,Z 625.096,A -85,B 0,C 180,E1 13580.871,E2 13580.871} C_VEL
LIN {X 0,Y 333.913,Z 630.136,A -85,B 0,C 180,E1 13585.926,E2 13585.926} C_VEL
LIN {X 0,Y 334.053,Z 631.422,A -85,B 0,C 180,E1 13589.996,E2 13589.996} C_VEL
LIN {X 0,Y 334.015,Z 629.337,A -85,B 0,C 180,E1 13595.197,E2 13595.197} C_VEL
LIN {X 0,Y 334.316,Z 622.115,A -85,B 0,C 180,E1 13601.092,E2 13601.092} C_VEL
LIN {X 0,Y 335.718,Z 609.355,A -85,B 0,C 180,E1 13607.041,E2 13607.041} C_VEL
LIN {X 0,Y 339.143,Z 590.129,A -85,B 0,C 180,E1 13612.988,E2 13612.988} C_VEL
LIN {X 0,Y 344.345,Z 566.37,A -85,B 0,C 180,E1 13618.208,E2 13618.208} C_VEL
LIN {X 0,Y 347.395,Z 552.992,A -85,B 0,C 180,E1 13620.504,E2 13620.504} C_VEL
LIN {X 0,Y 346.695,Z 540.944,A -85,B 0,C 180,E1 13622.608,E2 13622.608} C_VEL
LIN {X 0,Y 346.176,Z 528.148,A -85,B 0,C 180,E1 13624.584,E2 13624.584} C_VEL
LIN {X 0,Y 352.979,Z 496.342,A -85,B 0,C 180,E1 13627.865,E2 13627.865} C_VEL
LIN {X 0,Y 359.292,Z 460.344,A -85,B 0,C 180,E1 13630.375,E2 13630.375} C_VEL
LIN {X 0,Y 360.444,Z 447.126,A -85,B 0,C 180,E1 13631.112,E2 13631.112} C_VEL
LIN {X 0,Y 350.908,Z 420.296,A -85,B 0,C 180,E1 13633.974,E2 13633.974} C_VEL
LIN {X 0,Y 352.832,Z 409.141,A -85,B 0,C 180,E1 13636.044,E2 13636.044} C_VEL
LIN {X 0,Y 354.52,Z 414.452,A -85,B 0,C 180,E1 13639.815,E2 13639.815} C_VEL
LIN {X 0,Y 358.121,Z 424.293,A -85,B 0,C 180,E1 13642.516,E2 13642.516} C_VEL
LIN {X 0,Y 360.626,Z 438.942,A -85,B 0,C 180,E1 13644.71,E2 13644.71} C_VEL
LIN {X 0,Y 354.106,Z 473.452,A -85,B 0,C 180,E1 13647.331,E2 13647.331} C_VEL
LIN {X 0,Y 346.913,Z 505.365,A -85,B 0,C 180,E1 13650.946,E2 13650.946} C_VEL
LIN {X 0,Y 340.484,Z 530.361,A -85,B 0,C 180,E1 13655.012,E2 13655.012} C_VEL
LIN {X 0,Y 334.921,Z 550.946,A -85,B 0,C 180,E1 13659.837,E2 13659.837} C_VEL
LIN {X 0,Y 330.429,Z 566.586,A -85,B 0,C 180,E1 13665.403,E2 13665.403} C_VEL
LIN {X 0,Y 328.115,Z 575.352,A -85,B 0,C 180,E1 13670.705,E2 13670.705} C_VEL
LIN {X 0,Y 327.22,Z 578.516,A -85,B 0,C 180,E1 13674.689,E2 13674.689} C_VEL
LIN {X 0,Y 326.7,Z 578.625,A -85,B 0,C 180,E1 13679.998,E2 13679.998} C_VEL
LIN {X 0,Y 326.673,Z 573.794,A -85,B 0,C 180,E1 13685.316,E2 13685.316} C_VEL
LIN {X 0,Y 327.476,Z 563.849,A -85,B 0,C 180,E1 13690.655,E2 13690.655} C_VEL
LIN {X 0,Y 329.356,Z 547.799,A -85,B 0,C 180,E1 13696.008,E2 13696.008} C_VEL
LIN {X 0,Y 332.45,Z 526.017,A -85,B 0,C 180,E1 13700.951,E2 13700.951} C_VEL
LIN {X 0,Y 336.098,Z 500.411,A -85,B 0,C 180,E1 13705.068,E2 13705.068} C_VEL
LIN {X 0,Y 340.221,Z 469.474,A -85,B 0,C 180,E1 13708.576,E2 13708.576} C_VEL
LIN {X 0,Y 343.858,Z 435.059,A -85,B 0,C 180,E1 13711.2,E2 13711.2} C_VEL
LIN {X 0,Y 335.92,Z 405.147,A -85,B 0,C 180,E1 13713.377,E2 13713.377} C_VEL
LIN {X 0,Y 323.79,Z 370.16,A -85,B 0,C 180,E1 13715.58,E2 13715.58} C_VEL
LIN {X 0,Y 323.703,Z 370.16,A -85,B 0,C 180,E1 13724.547,E2 13724.547} C_VEL
LIN {X 0,Y 323.724,Z 370.838,A -85,B 0,C 180,E1 13725.148,E2 13725.148} C_VEL
LIN {X 0,Y 326.434,Z 376.144,A -85,B 0,C 180,E1 13725.82,E2 13725.82} C_VEL
LIN {X 0,Y 344.211,Z 407.904,A -85,B 0,C 180,E1 13729.954,E2 13729.954} C_VEL
LIN {X 0,Y 355.494,Z 436.79,A -85,B 0,C 180,E1 13733.405,E2 13733.405} C_VEL
LIN {X 0,Y 358.891,Z 451.437,A -85,B 0,C 180,E1 13735.093,E2 13735.093} C_VEL
LIN {X 0,Y 352.561,Z 482.883,A -85,B 0,C 180,E1 13737.905,E2 13737.905} C_VEL
LIN {X 0,Y 345.521,Z 510.547,A -85,B 0,C 180,E1 13741.547,E2 13741.547} C_VEL
LIN {X 0,Y 338.737,Z 533.601,A -85,B 0,C 180,E1 13745.936,E2 13745.936} C_VEL
LIN {X 0,Y 333.393,Z 551.43,A -85,B 0,C 180,E1 13750.783,E2 13750.783} C_VEL
LIN {X 0,Y 329.239,Z 565.888,A -85,B 0,C 180,E1 13756.712,E2 13756.712} C_VEL
LIN {X 0,Y 327.385,Z 573.73,A -85,B 0,C 180,E1 13762.03,E2 13762.03} C_VEL
LIN {X 0,Y 326.494,Z 577.491,A -85,B 0,C 180,E1 13767.346,E2 13767.346} C_VEL
LIN {X 0,Y 326.512,Z 577.448,A -85,B 0,C 180,E1 13772.662,E2 13772.662} C_VEL
LIN {X 0,Y 327.436,Z 573.601,A -85,B 0,C 180,E1 13777.977,E2 13777.977} C_VEL
LIN {X 0,Y 329.64,Z 564.42,A -85,B 0,C 180,E1 13783.956,E2 13783.956} C_VEL
LIN {X 0,Y 334.084,Z 549.02,A -85,B 0,C 180,E1 13789.873,E2 13789.873} C_VEL
LIN {X 0,Y 340.113,Z 528.774,A -85,B 0,C 180,E1 13795.02,E2 13795.02} C_VEL
LIN {X 0,Y 347.187,Z 504.237,A -85,B 0,C 180,E1 13799.3,E2 13799.3} C_VEL
LIN {X 0,Y 353.997,Z 476.256,A -85,B 0,C 180,E1 13802.683,E2 13802.683} C_VEL
LIN {X 0,Y 358.779,Z 448.908,A -85,B 0,C 180,E1 13805.034,E2 13805.034} C_VEL
LIN {X 0,Y 349.504,Z 420.03,A -85,B 0,C 180,E1 13808.466,E2 13808.466} C_VEL
LIN {X 0,Y 335.761,Z 391.943,A -85,B 0,C 180,E1 13811.932,E2 13811.932} C_VEL
LIN {X 0,Y 323.787,Z 371.589,A -85,B 0,C 180,E1 13814.688,E2 13814.688} C_VEL
LIN {X 0,Y 323.643,Z 370.16,A -85,B 0,C 180,E1 13814.858,E2 13814.858} C_VEL
LIN {X 0,Y 323.576,Z 370.16,A -85,B 0,C 180,E1 13822.698,E2 13822.698} C_VEL
LIN {X 0,Y 323.709,Z 370.16,A -85,B 0,C 180,E1 13829.042,E2 13829.042} C_VEL
LIN {X 0,Y 323.969,Z 370.16,A -85,B 0,C 180,E1 13835.131,E2 13835.131} C_VEL
LIN {X 0,Y 324.342,Z 370.16,A -85,B 0,C 180,E1 13840.931,E2 13840.931} C_VEL
LIN {X 0,Y 324.714,Z 370.16,A -85,B 0,C 180,E1 13848.283,E2 13848.283} C_VEL
LIN {X 0,Y 325.198,Z 370.16,A -85,B 0,C 180,E1 13854.659,E2 13854.659} C_VEL
LIN {X 0,Y 325.55,Z 370.16,A -85,B 0,C 180,E1 13860.002,E2 13860.002} C_VEL
LIN {X 0,Y 324.968,Z 370.16,A -85,B 0,C 180,E1 13868.036,E2 13868.036} C_VEL
LIN {X 0,Y 324.465,Z 370.16,A -85,B 0,C 180,E1 13876.259,E2 13876.259} C_VEL
LIN {X 0,Y 324.154,Z 370.16,A -85,B 0,C 180,E1 13881.941,E2 13881.941} C_VEL
LIN {X 0,Y 323.892,Z 370.16,A -85,B 0,C 180,E1 13887.868,E2 13887.868} C_VEL
LIN {X 0,Y 323.667,Z 370.16,A -85,B 0,C 180,E1 13894.147,E2 13894.147} C_VEL
LIN {X 0,Y 323.674,Z 370.16,A -85,B 0,C 180,E1 13900.04,E2 13900.04} C_VEL
LIN {X 0,Y 326.131,Z 375.852,A -85,B 0,C 180,E1 13900.738,E2 13900.738} C_VEL
LIN {X 0,Y 344.582,Z 408.18,A -85,B 0,C 180,E1 13904.873,E2 13904.873} C_VEL
LIN {X 0,Y 357.987,Z 439.936,A -85,B 0,C 180,E1 13908.165,E2 13908.165} C_VEL
LIN {X 0,Y 360.64,Z 450.499,A -85,B 0,C 180,E1 13909.132,E2 13909.132} C_VEL
LIN {X 0,Y 354.789,Z 486.854,A -85,B 0,C 180,E1 13911.382,E2 13911.382} C_VEL
LIN {X 0,Y 347.754,Z 520.999,A -85,B 0,C 180,E1 13914.576,E2 13914.576} C_VEL
LIN {X 0,Y 340.585,Z 551.483,A -85,B 0,C 180,E1 13918.696,E2 13918.696} C_VEL
LIN {X 0,Y 334.401,Z 576.857,A -85,B 0,C 180,E1 13923.44,E2 13923.44} C_VEL
LIN {X 0,Y 329.776,Z 598.124,A -85,B 0,C 180,E1 13928.93,E2 13928.93} C_VEL
LIN {X 0,Y 327.233,Z 613.555,A -85,B 0,C 180,E1 13934.568,E2 13934.568} C_VEL
LIN {X 0,Y 326.266,Z 624.445,A -85,B 0,C 180,E1 13940.649,E2 13940.649} C_VEL
LIN {X 0,Y 326.129,Z 628.682,A -85,B 0,C 180,E1 13944.669,E2 13944.669} C_VEL
LIN {X 0,Y 326.191,Z 630.786,A -85,B 0,C 180,E1 13949.996,E2 13949.996} C_VEL
LIN {X 0,Y 326.124,Z 628.695,A -85,B 0,C 180,E1 13955.323,E2 13955.323} C_VEL
LIN {X 0,Y 326.459,Z 621.471,A -85,B 0,C 180,E1 13961.355,E2 13961.355} C_VEL
LIN {X 0,Y 327.978,Z 608.676,A -85,B 0,C 180,E1 13967.456,E2 13967.456} C_VEL
LIN {X 0,Y 331.656,Z 589.422,A -85,B 0,C 180,E1 13973.537,E2 13973.537} C_VEL
LIN {X 0,Y 337.07,Z 566.008,A -85,B 0,C 180,E1 13978.79,E2 13978.79} C_VEL
LIN {X 0,Y 343.88,Z 537.782,A -85,B 0,C 180,E1 13983.345,E2 13983.345} C_VEL
LIN {X 0,Y 346.176,Z 528.148,A -85,B 0,C 180,E1 13984.584,E2 13984.584} C_VEL
LIN {X 0,Y 345.664,Z 514.786,A -85,B 0,C 180,E1 13986.477,E2 13986.477} C_VEL
LIN {X 0,Y 345.112,Z 502.688,A -85,B 0,C 180,E1 13988.037,E2 13988.037} C_VEL
LIN {X 0,Y 345.478,Z 500.812,A -85,B 0,C 180,E1 13988.213,E2 13988.213} C_VEL
LIN {X 0,Y 352.082,Z 466.099,A -85,B 0,C 180,E1 13990.811,E2 13990.811} C_VEL
LIN {X 0,Y 354.116,Z 450.03,A -85,B 0,C 180,E1 13991.741,E2 13991.741} C_VEL
LIN {X 0,Y 348.048,Z 430.996,A -85,B 0,C 180,E1 13993.88,E2 13993.88} C_VEL
LIN {X 0,Y 350.714,Z 417.058,A -85,B 0,C 180,E1 13996.48,E2 13996.48} C_VEL
LIN {X 0,Y 352.108,Z 422.36,A -85,B 0,C 180,E1 13999.714,E2 13999.714} C_VEL
LIN {X 0,Y 354.691,Z 431.552,A -85,B 0,C 180,E1 14002.186,E2 14002.186} C_VEL
LIN {X 0,Y 355.793,Z 442.393,A -85,B 0,C 180,E1 14003.838,E2 14003.838} C_VEL
LIN {X 0,Y 348.488,Z 476.504,A -85,B 0,C 180,E1 14006.551,E2 14006.551} C_VEL
LIN {X 0,Y 340.812,Z 507.264,A -85,B 0,C 180,E1 14010.174,E2 14010.174} C_VEL
LIN {X 0,Y 333.653,Z 532.672,A -85,B 0,C 180,E1 14014.464,E2 14014.464} C_VEL
LIN {X 0,Y 327.702,Z 552.667,A -85,B 0,C 180,E1 14019.373,E2 14019.373} C_VEL
LIN {X 0,Y 323.323,Z 566.483,A -85,B 0,C 180,E1 14024.379,E2 14024.379} C_VEL
LIN {X 0,Y 320.927,Z 574.729,A -85,B 0,C 180,E1 14029.122,E2 14029.122} C_VEL
LIN {X 0,Y 319.392,Z 579.401,A -85,B 0,C 180,E1 14034.558,E2 14034.558} C_VEL
LIN {X 0,Y 318.821,Z 579.24,A -85,B 0,C 180,E1 14039.998,E2 14039.998} C_VEL
LIN {X 0,Y 318.871,Z 573.236,A -85,B 0,C 180,E1 14046.13,E2 14046.13} C_VEL
LIN {X 0,Y 319.868,Z 562.232,A -85,B 0,C 180,E1 14051.602,E2 14051.602} C_VEL
LIN {X 0,Y 322.013,Z 544.948,A -85,B 0,C 180,E1 14057.086,E2 14057.086} C_VEL
LIN {X 0,Y 325.215,Z 523.134,A -85,B 0,C 180,E1 14061.862,E2 14061.862} C_VEL
LIN {X 0,Y 329.163,Z 496.212,A -85,B 0,C 180,E1 14066.054,E2 14066.054} C_VEL
LIN {X 0,Y 333.321,Z 465.525,A -85,B 0,C 180,E1 14069.41,E2 14069.41} C_VEL
LIN {X 0,Y 336.29,Z 433.473,A -85,B 0,C 180,E1 14071.825,E2 14071.825} C_VEL
LIN {X 0,Y 325.959,Z 399.054,A -85,B 0,C 180,E1 14074.375,E2 14074.375} C_VEL
LIN {X 0,Y 315.833,Z 370.16,A -85,B 0,C 180,E1 14076.228,E2 14076.228} C_VEL
LIN {X 0,Y 315.659,Z 370.16,A -85,B 0,C 180,E1 14083.497,E2 14083.497} C_VEL
LIN {X 0,Y 317.953,Z 375.659,A -85,B 0,C 180,E1 14084.158,E2 14084.158} C_VEL
LIN {X 0,Y 334.499,Z 403.467,A -85,B 0,C 180,E1 14088.187,E2 14088.187} C_VEL
LIN {X 0,Y 346.676,Z 431.96,A -85,B 0,C 180,E1 14091.815,E2 14091.815} C_VEL
LIN {X 0,Y 352.488,Z 452.567,A -85,B 0,C 180,E1 14094.373,E2 14094.373} C_VEL
LIN {X 0,Y 345.928,Z 483.698,A -85,B 0,C 180,E1 14097.213,E2 14097.213} C_VEL
LIN {X 0,Y 338.62,Z 511.274,A -85,B 0,C 180,E1 14100.913,E2 14100.913} C_VEL
LIN {X 0,Y 331.53,Z 534.287,A -85,B 0,C 180,E1 14105.378,E2 14105.378} C_VEL
LIN {X 0,Y 325.908,Z 552.096,A -85,B 0,C 180,E1 14110.323,E2 14110.323} C_VEL
LIN {X 0,Y 321.542,Z 566.535,A -85,B 0,C 180,E1 14116.388,E2 14116.388} C_VEL
LIN {X 0,Y 319.577,Z 574.369,A -85,B 0,C 180,E1 14121.834,E2 14121.834} C_VEL
LIN {X 0,Y 318.625,Z 578.129,A -85,B 0,C 180,E1 14127.281,E2 14127.281} C_VEL
LIN {X 0,Y 318.645,Z 578.086,A -85,B 0,C 180,E1 14132.727,E2 14132.727} C_VEL
LIN {X 0,Y 319.622,Z 574.243,A -85,B 0,C 180,E1 14138.173,E2 14138.173} C_VEL
LIN {X 0,Y 321.953,Z 565.142,A -85,B 0,C 180,E1 14144.258,E2 14144.258} C_VEL
LIN {X 0,Y 326.307,Z 550.718,A -85,B 0,C 180,E1 14150.013,E2 14150.013} C_VEL
LIN {X 0,Y 332.557,Z 531.006,A -85,B 0,C 180,E1 14155.268,E2 14155.268} C_VEL
LIN {X 0,Y 339.796,Z 506.79,A -85,B 0,C 180,E1 14159.676,E2 14159.676} C_VEL
LIN {X 0,Y 347.117,Z 478.622,A -85,B 0,C 180,E1 14163.228,E2 14163.228} C_VEL
LIN {X 0,Y 352.206,Z 451.488,A -85,B 0,C 180,E1 14165.648,E2 14165.648} C_VEL
LIN {X 0,Y 343.482,Z 423.381,A -85,B 0,C 180,E1 14169.144,E2 14169.144} C_VEL
LIN {X 0,Y 329.408,Z 394.276,A -85,B 0,C 180,E1 14172.949,E2 14172.949} C_VEL
LIN {X 0,Y 317.59,Z 375.294,A -85,B 0,C 180,E1 14175.797,E2 14175.797} C_VEL
LIN {X 0,Y 315.611,Z 370.16,A -85,B 0,C 180,E1 14176.381,E2 14176.381} C_VEL
LIN {X 0,Y 315.597,Z 370.16,A -85,B 0,C 180,E1 14184.858,E2 14184.858} C_VEL
LIN {X 0,Y 315.85,Z 370.16,A -85,B 0,C 180,E1 14191.362,E2 14191.362} C_VEL
LIN {X 0,Y 316.158,Z 370.16,A -85,B 0,C 180,E1 14197.478,E2 14197.478} C_VEL
LIN {X 0,Y 316.575,Z 370.16,A -85,B 0,C 180,E1 14203.328,E2 14203.328} C_VEL
LIN {X 0,Y 317.028,Z 370.16,A -85,B 0,C 180,E1 14211.765,E2 14211.765} C_VEL
LIN {X 0,Y 317.671,Z 370.16,A -85,B 0,C 180,E1 14220.002,E2 14220.002} C_VEL
LIN {X 0,Y 317.02,Z 370.16,A -85,B 0,C 180,E1 14228.239,E2 14228.239} C_VEL
LIN {X 0,Y 316.467,Z 370.16,A -85,B 0,C 180,E1 14236.895,E2 14236.895} C_VEL
LIN {X 0,Y 316.033,Z 370.16,A -85,B 0,C 180,E1 14245.541,E2 14245.541} C_VEL
LIN {X 0,Y 315.767,Z 370.16,A -85,B 0,C 180,E1 14251.831,E2 14251.831} C_VEL
LIN {X 0,Y 315.751,Z 370.16,A -85,B 0,C 180,E1 14258.481,E2 14258.481} C_VEL
LIN {X 0,Y 318.217,Z 375.896,A -85,B 0,C 180,E1 14259.208,E2 14259.208} C_VEL
